  MoveL 5113 to (559.6, 473.58, 88) mm, rotated rx -180 ry 0 rz 160 deg; joints [2.536, 74.611, -25.018, -151.413, 53.222, 161.93]
  Set speed (17.9 mm/s)
  Call Extruder(373.72184)
  MoveL 5114 to (560.12, 474.8, 88) mm, rotated rx -180 ry 0 rz 160 deg; joints [2.67, 74.736, -25.273, -151.206, 53.149, 161.757]
  Set speed (17.9 mm/s)
  Call Extruder(378.01849)
  MoveL 5115 to (560.64, 476.06, 88) mm, rotated rx 180 ry 0 rz 160 deg; joints [2.809, 74.862, -25.532, -150.994, 53.077, 161.578]
  Set speed (17.9 mm/s)
  Call Extruder(382.11956)
  MoveL 5116 to (561.1, 477.28, 88) mm, rotated rx -180 ry 0 rz 160 deg; joints [2.943, 74.976, -25.765, -150.791, 53.016, 161.41]
  Set speed (17.9 mm/s)
  Call Extruder(386.18215)
  MoveL 5117 to (561.55, 478.49, 88) mm, rotated rx -180 ry 0 rz 160 deg; joints [3.076, 75.088, -25.993, -150.59, 52.957, 161.244]
  Call Extruder(390.52183)
  MoveL 5118 to (561.98, 479.8, 88) mm, rotated rx 180 ry 0 rz 160 deg; joints [3.219, 75.2, -26.222, -150.377, 52.902, 161.069]
  Set speed (17.9 mm/s)
  Call Extruder(394.64842)
  MoveL 5119 to (562.38, 481.05, 88) mm, rotated rx -180 ry 0 rz 160 deg; joints [3.356, 75.305, -26.435, -150.174, 52.852, 160.904]
  Set speed (17.9 mm/s)
  Call Extruder(398.90970)
  MoveL 5120 to (562.75, 482.35, 88) mm, rotated rx 180 ry 0 rz 160 deg; joints [3.499, 75.405, -26.64, -149.965, 52.808, 160.736]
  Set speed (17.9 mm/s)
  Call Extruder(402.92421)
  MoveL 5121 to (563.09, 483.58, 88) mm, rotated rx -180 ry 0 rz 160 deg; joints [3.633, 75.498, -26.83, -149.769, 52.769, 160.579]
  Call Extruder(407.31030)
  MoveL 5122 to (563.42, 484.93, 88) mm, rotated rx 180 ry 0 rz 160 deg; joints [3.781, 75.593, -27.022, -149.556, 52.735, 160.411]
  Set speed (17.9 mm/s)
  Call Extruder(411.41596)
  MoveL 5123 to (563.72, 486.2, 88) mm, rotated rx 180 ry 0 rz 160 deg; joints [3.92, 75.678, -27.196, -149.357, 52.705, 160.254]
  Set speed (17.9 mm/s)
  Call Extruder(419.87700)
  MoveL 5124 to (564.23, 488.84, 88) mm, rotated rx -180 ry 0 rz 160 deg; joints [4.21, 75.838, -27.52, -148.951, 52.662, 159.941]
  Set speed (17.9 mm/s)
  Call Extruder(428.25790)
  MoveL 5125 to (564.64, 491.48, 88) mm, rotated rx -180 ry 0 rz 160 deg; joints [4.499, 75.975, -27.801, -148.553, 52.64, 159.641]
  Call Extruder(436.73506)
  MoveL 5126 to (564.94, 494.16, 88) mm, rotated rx 180 ry 0 rz 160 deg; joints [4.793, 76.093, -28.041, -148.158, 52.639, 159.35]
  Call Extruder(445.02927)
  MoveL 5127 to (565.12, 496.79, 88) mm, rotated rx 180 ry 0 rz 160 deg; joints [5.082, 76.188, -28.232, -147.778, 52.659, 159.079]
  Call Extruder(453.41460)
  MoveL 5128 to (565.2, 499.45, 88) mm, rotated rx -180 ry 0 rz 160 deg; joints [5.376, 76.262, -28.384, -147.402, 52.7, 158.818]
  Set speed (18.0 mm/s)
  Call Extruder(461.67884)
  MoveL 5129 to (565.16, 502.08, 88) mm, rotated rx -180 ry 0 rz 160 deg; joints [5.666, 76.314, -28.488, -147.04, 52.761, 158.576]
  Set speed (17.9 mm/s)
  Call Extruder(470.17572)
  MoveL 5130 to (565.02, 504.78, 88) mm, rotated rx -180 ry 0 rz 160 deg; joints [5.965, 76.345, -28.551, -146.678, 52.844, 158.343]
  Call Extruder(478.48137)
  MoveL 5131 to (564.77, 507.41, 88) mm, rotated rx 180 ry 0 rz 160 deg; joints [6.258, 76.352, -28.566, -146.334, 52.946, 158.132]
  Set speed (18.0 mm/s)
  Call Extruder(487.03739)
  MoveL 5132 to (564.41, 510.11, 88) mm, rotated rx 180 ry 0 rz 160 deg; joints [6.559, 76.338, -28.536, -145.99, 53.071, 157.932]
  Call Extruder(495.31907)
  MoveL 5133 to (563.95, 512.71, 88) mm, rotated rx 180 ry 0 rz 160 deg; joints [6.851, 76.302, -28.464, -145.668, 53.212, 157.755]
  Set speed (17.9 mm/s)
  Call Extruder(503.76190)
  MoveL 5134 to (563.37, 515.33, 88) mm, rotated rx 180 ry 0 rz 160 deg; joints [7.147, 76.243, -28.344, -145.352, 53.374, 157.594]
  Set speed (17.9 mm/s)
  Call Extruder(507.92287)
  MoveL 5135 to (563.04, 516.61, 88) mm, rotated rx -180 ry 0 rz 160 deg; joints [7.293, 76.204, -28.266, -145.201, 53.463, 157.522]
  Set speed (17.9 mm/s)
  Call Extruder(512.03156)
  MoveL 5136 to (562.7, 517.87, 88) mm, rotated rx -180 ry 0 rz 160 deg; joints [7.436, 76.164, -28.183, -145.054, 53.552, 157.454]
  Set speed (17.9 mm/s)
  Call Extruder(516.36211)
  MoveL 5137 to (562.3, 519.18, 88) mm, rotated rx 180 ry 0 rz 160 deg; joints [7.587, 76.113, -28.08, -144.904, 53.653, 157.389]
  Set speed (17.9 mm/s)
  Call Extruder(520.51999)
  MoveL 5138 to (561.91, 520.44, 88) mm, rotated rx 180 ry 0 rz 160 deg; joints [7.731, 76.061, -27.975, -144.76, 53.752, 157.329]
  Set speed (17.9 mm/s)
  Call Extruder(528.91386)
  MoveL 5139 to (561.02, 522.96, 88) mm, rotated rx 180 ry 0 rz 160 deg; joints [8.022, 75.938, -27.725, -144.482, 53.968, 157.224]
  Set speed (17.9 mm/s)
  Call Extruder(533.10830)
  MoveL 5140 to (560.53, 524.2, 88) mm, rotated rx -180 ry 0 rz 160 deg; joints [8.166, 75.868, -27.582, -144.349, 54.083, 157.18]
  Set speed (17.9 mm/s)
  Call Extruder(537.31700)
  MoveL 5141 to (560.03, 525.44, 88) mm, rotated rx -180 ry 0 rz 160 deg; joints [8.311, 75.795, -27.433, -144.216, 54.2, 157.138]
  Set speed (17.9 mm/s)
  Call Extruder(541.50408)
  MoveL 5142 to (559.49, 526.66, 88) mm, rotated rx 180 ry 0 rz 160 deg; joints [8.453, 75.714, -27.269, -144.09, 54.323, 157.104]
  Set speed (17.9 mm/s)
  Call Extruder(545.52808)
  MoveL 5143 to (558.96, 527.82, 88) mm, rotated rx 180 ry 0 rz 160 deg; joints [8.59, 75.635, -27.107, -143.969, 54.443, 157.073]
  Set speed (17.9 mm/s)
  Call Extruder(548.70706)
  MoveL 5144 to (558.53, 528.73, 88) mm, rotated rx 180 ry 0 rz 160 deg; joints [8.698, 75.568, -26.972, -143.876, 54.541, 157.052]
  Set speed (17.9 mm/s)
  Call Extruder(554.38655)
  MoveL 5145 to (557.71, 530.34, 88) mm, rotated rx 180 ry 0 rz 160 deg; joints [8.889, 75.442, -26.714, -143.715, 54.721, 157.022]
  Set speed (18.0 mm/s)
  Call Extruder(558.28991)
  MoveL 5146 to (557.12, 531.43, 88) mm, rotated rx -180 ry 0 rz 160 deg; joints [9.02, 75.349, -26.526, -143.608, 54.85, 157.007]
  Set speed (17.9 mm/s)
  Call Extruder(562.42698)
  MoveL 5147 to (556.47, 532.58, 88) mm, rotated rx -180 ry 0 rz 160 deg; joints [9.158, 75.248, -26.319, -143.497, 54.989, 156.994]
  Set speed (18.0 mm/s)
  Call Extruder(566.58221)
  MoveL 5148 to (555.8, 533.72, 88) mm, rotated rx -180 ry 0 rz 160 deg; joints [9.296, 75.141, -26.102, -143.388, 55.131, 156.986]
  Call Extruder(570.79001)
  MoveL 5149 to (555.1, 534.86, 88) mm, rotated rx -180 ry 0 rz 160 deg; joints [9.435, 75.028, -25.872, -143.281, 55.28, 156.982]
  Set speed (17.9 mm/s)
  Call Extruder(574.99054)
  MoveL 5150 to (554.37, 535.98, 88) mm, rotated rx 180 ry 0 rz 160 deg; joints [9.572, 74.912, -25.633, -143.178, 55.431, 156.984]
  Set speed (17.9 mm/s)
  Call Extruder(579.19251)
  MoveL 5151 to (553.62, 537.08, 88) mm, rotated rx 180 ry 0 rz 160 deg; joints [9.709, 74.791, -25.387, -143.077, 55.585, 156.989]
  Set speed (17.9 mm/s)
  Call Extruder(583.43346)
  MoveL 5152 to (552.85, 538.19, 88) mm, rotated rx 180 ry 0 rz 160 deg; joints [9.846, 74.665, -25.129, -142.979, 55.744, 156.999]
  Call Extruder(587.57525)
  MoveL 5153 to (552.06, 539.24, 88) mm, rotated rx -180 ry 0 rz 160 deg; joints [9.978, 74.537, -24.867, -142.886, 55.902, 157.013]
  Set speed (17.9 mm/s)
  Call Extruder(591.76685)
  MoveL 5154 to (551.25, 540.3, 88) mm, rotated rx 180 ry 0 rz 160 deg; joints [10.111, 74.405, -24.597, -142.794, 56.064, 157.031]
  Call Extruder(595.94820)
  MoveL 5155 to (550.42, 541.34, 88) mm, rotated rx 180 ry 0 rz 160 deg; joints [10.243, 74.268, -24.317, -142.707, 56.229, 157.054]
  Set speed (17.9 mm/s)
  Call Extruder(600.26743)
  MoveL 5156 to (549.53, 542.39, 88) mm, rotated rx 180 ry 0 rz 160 deg; joints [10.377, 74.124, -24.021, -142.619, 56.403, 157.082]
  Set speed (17.9 mm/s)
  Call Extruder(604.33296)
  MoveL 5157 to (548.68, 543.36, 88) mm, rotated rx 180 ry 0 rz 160 deg; joints [10.503, 73.984, -23.734, -142.539, 56.568, 157.113]
  Set speed (17.9 mm/s)
  Call Extruder(608.56191)
  MoveL 5158 to (547.78, 544.36, 88) mm, rotated rx 180 ry 0 rz 160 deg; joints [10.633, 73.835, -23.429, -142.459, 56.742, 157.148]
  Set speed (17.9 mm/s)
  Call Extruder(612.71555)
  MoveL 5159 to (546.87, 545.32, 88) mm, rotated rx -180 ry 0 rz 160 deg; joints [10.759, 73.686, -23.123, -142.383, 56.916, 157.187]
  Set speed (17.9 mm/s)
  Call Extruder(616.93142)
  MoveL 5160 to (545.93, 546.27, 88) mm, rotated rx 180 ry 0 rz 160 deg; joints [10.885, 73.531, -22.805, -142.309, 57.094, 157.23]
  Set speed (18.0 mm/s)
  Call Extruder(621.11476)
  MoveL 5161 to (544.98, 547.2, 88) mm, rotated rx 180 ry 0 rz 160 deg; joints [11.009, 73.374, -22.482, -142.238, 57.273, 157.277]
  Set speed (17.9 mm/s)
  Call Extruder(625.39673)
  MoveL 5162 to (543.98, 548.13, 88) mm, rotated rx 180 ry 0 rz 160 deg; joints [11.135, 73.21, -22.144, -142.168, 57.459, 157.329]
  Set speed (17.9 mm/s)
  Call Extruder(629.55539)
  MoveL 5163 to (543, 549.01, 88) mm, rotated rx -180 ry 0 rz 160 deg; joints [11.255, 73.048, -21.81, -142.104, 57.641, 157.383]
  Set speed (17.9 mm/s)
  Call Extruder(633.66255)
  MoveL 5164 to (542, 549.86, 88) mm, rotated rx 180 ry 0 rz 160 deg; joints [11.373, 72.885, -21.474, -142.042, 57.823, 157.44]
  Call Extruder(637.94036)
  MoveL 5165 to (540.96, 550.73, 88) mm, rotated rx 180 ry 0 rz 160 deg; joints [11.494, 72.712, -21.118, -141.981, 58.013, 157.503]
  Set speed (17.9 mm/s)
  Call Extruder(642.04901)
  MoveL 5166 to (539.93, 551.54, 88) mm, rotated rx 180 ry 0 rz 160 deg; joints [11.608, 72.544, -20.771, -141.925, 58.198, 157.567]
  Call Extruder(646.27944)
  MoveL 5167 to (538.86, 552.35, 88) mm, rotated rx 180 ry 0 rz 160 deg; joints [11.725, 72.368, -20.407, -141.87, 58.39, 157.637]
  Set speed (17.9 mm/s)
  Call Extruder(650.48406)
  MoveL 5168 to (537.78, 553.14, 88) mm, rotated rx -180 ry 0 rz 160 deg; joints [11.839, 72.191, -20.041, -141.818, 58.582, 157.709]
  Call Extruder(654.65527)
  MoveL 5169 to (536.69, 553.89, 88) mm, rotated rx 180 ry 0 rz 160 deg; joints [11.95, 72.013, -19.672, -141.769, 58.774, 157.785]
  Set speed (17.9 mm/s)
  Call Extruder(658.83011)
  MoveL 5170 to (535.58, 554.63, 88) mm, rotated rx 180 ry 0 rz 160 deg; joints [12.06, 71.832, -19.299, -141.723, 58.967, 157.863]
  Set speed (17.9 mm/s)
  Call Extruder(663.02238)
  MoveL 5171 to (534.46, 555.35, 88) mm, rotated rx 180 ry 0 rz 160 deg; joints [12.168, 71.649, -18.919, -141.679, 59.162, 157.945]
  Set speed (17.9 mm/s)
  Call Extruder(667.21459)
  MoveL 5172 to (533.32, 556.04, 88) mm, rotated rx -180 ry 0 rz 160 deg; joints [12.274, 71.464, -18.535, -141.638, 59.358, 158.03]
  Set speed (18.0 mm/s)
  Call Extruder(671.40809)
  MoveL 5173 to (532.17, 556.71, 88) mm, rotated rx -180 ry 0 rz 160 deg; joints [12.379, 71.276, -18.145, -141.599, 59.556, 158.118]
  Set speed (17.9 mm/s)
  Call Extruder(675.05317)
  MoveL 5174 to (531.15, 557.28, 88) mm, rotated rx 180 ry 0 rz 160 deg; joints [12.468, 71.112, -17.804, -141.567, 59.728, 158.197]
  Set speed (17.9 mm/s)
  Call Extruder(679.85489)
  MoveL 5175 to (529.8, 557.99, 88) mm, rotated rx -180 ry 0 rz 160 deg; joints [12.584, 70.894, -17.349, -141.529, 59.955, 158.305]
  Set speed (17.9 mm/s)
  Call Extruder(684.04696)
  MoveL 5176 to (528.61, 558.59, 88) mm, rotated rx -180 ry 0 rz 160 deg; joints [12.682, 70.701, -16.948, -141.498, 60.155, 158.402]
  Set speed (17.9 mm/s)
  Call Extruder(688.17169)
  MoveL 5177 to (527.43, 559.15, 88) mm, rotated rx -180 ry 0 rz 160 deg; joints [12.777, 70.51, -16.55, -141.47, 60.352, 158.5]
  Set speed (17.9 mm/s)
  Call Extruder(692.46193)
  MoveL 5178 to (526.18, 559.7, 88) mm, rotated rx -180 ry 0 rz 160 deg; joints [12.873, 70.31, -16.132, -141.444, 60.557, 158.606]
  Set speed (17.9 mm/s)
  Call Extruder(696.56563)
  MoveL 5179 to (524.99, 560.22, 88) mm, rotated rx -180 ry 0 rz 160 deg; joints [12.964, 70.118, -15.731, -141.421, 60.754, 158.708]
  Set speed (17.9 mm/s)
  Call Extruder(700.85853)
  MoveL 5180 to (523.72, 560.72, 88) mm, rotated rx -180 ry 0 rz 160 deg; joints [13.055, 69.915, -15.306, -141.4, 60.96, 158.819]
  Set speed (17.9 mm/s)
  Call Extruder(704.88381)
  MoveL 5181 to (522.52, 561.18, 88) mm, rotated rx -180 ry 0 rz 160 deg; joints [13.14, 69.725, -14.907, -141.382, 61.154, 158.924]
  Set speed (17.9 mm/s)
  Call Extruder(709.30941)
  MoveL 5182 to (521.2, 561.65, 88) mm, rotated rx -180 ry 0 rz 160 deg; joints [13.229, 69.513, -14.464, -141.366, 61.367, 159.043]
  Set speed (17.9 mm/s)
  Call Extruder(713.41630)
  MoveL 5183 to (519.97, 562.07, 88) mm, rotated rx 180 ry 0 rz 160 deg; joints [13.311, 69.317, -14.053, -141.352, 61.564, 159.154]
  Call Extruder(717.65007)
  MoveL 5184 to (518.68, 562.46, 88) mm, rotated rx -180 ry 0 rz 160 deg; joints [13.392, 69.113, -13.624, -141.342, 61.768, 159.273]
  Set speed (17.9 mm/s)
  Call Extruder(721.92491)
  MoveL 5185 to (517.38, 562.84, 88) mm, rotated rx -180 ry 0 rz 160 deg; joints [13.472, 68.907, -13.191, -141.332, 61.974, 159.394]
  Set speed (17.9 mm/s)
  Call Extruder(725.52012)
  MoveL 5186 to (516.27, 563.13, 88) mm, rotated rx -180 ry 0 rz 160 deg; joints [13.537, 68.733, -12.823, -141.328, 62.148, 159.498]
  Set speed (17.9 mm/s)
  Call Extruder(730.10548)
  MoveL 5187 to (514.86, 563.48, 88) mm, rotated rx 180 ry 0 rz 160 deg; joints [13.618, 68.511, -12.355, -141.323, 62.368, 159.632]
  Set speed (17.9 mm/s)
  Call Extruder(738.64656)
  MoveL 5188 to (512.2, 564.04, 88) mm, rotated rx -180 ry 0 rz 160 deg; joints [13.759, 68.094, -11.474, -141.324, 62.779, 159.89]
  Set speed (17.9 mm/s)
  Call Extruder(747.08753)
  MoveL 5189 to (509.56, 564.49, 88) mm, rotated rx 180 ry 0 rz 160 deg; joints [13.888, 67.681, -10.599, -141.335, 63.184, 160.152]
  Call Extruder(755.39717)
  MoveL 5190 to (506.93, 564.83, 88) mm, rotated rx 180 ry 0 rz 160 deg; joints [14.004, 67.273, -9.734, -141.356, 63.58, 160.417]
  Set speed (17.9 mm/s)
  Call Extruder(763.82579)
  MoveL 5191 to (504.26, 565.06, 88) mm, rotated rx 180 ry 0 rz 160 deg; joints [14.111, 66.86, -8.855, -141.388, 63.98, 160.692]
  Set speed (18.0 mm/s)
  Call Extruder(772.24871)
  MoveL 5192 to (501.59, 565.18, 88) mm, rotated rx -180 ry 0 rz 160 deg; joints [14.206, 66.448, -7.974, -141.429, 64.377, 160.973]
  Set speed (17.9 mm/s)
  Call Extruder(780.47163)
  MoveL 5193 to (498.97, 565.19, 88) mm, rotated rx 180 ry 0 rz 160 deg; joints [14.286, 66.046, -7.115, -141.48, 64.761, 161.252]
  Set speed (10.0 mm/s)
  MoveL 5194 to (498.97, 565.19, 92) mm, rotated rx 180 ry 0 rz 160 deg; joints [14.286, 65.4, -6.792, -141.385, 64.508, 161.029]
  Set speed (120.0 mm/s)
  MoveL 5195 to (498.97, 565.42, 92) mm, rotated rx 180 ry 0 rz 160 deg; joints [14.315, 65.408, -6.81, -141.352, 64.51, 161.01]
  Set speed (18.0 mm/s)
  Call Extruder(789.01663)
  MoveL 5196 to (496.25, 565.32, 92) mm, rotated rx 180 ry 0 rz 160 deg; joints [14.386, 64.991, -5.919, -141.417, 64.903, 161.305]
  Call Extruder(797.44924)
  MoveL 5197 to (493.57, 565.11, 92) mm, rotated rx 180 ry 0 rz 160 deg; joints [14.444, 64.581, -5.043, -141.491, 65.286, 161.6]
  Set speed (18.0 mm/s)
  Call Extruder(805.77515)
  MoveL 5198 to (490.93, 564.8, 92) mm, rotated rx -180 ry 0 rz 160 deg; joints [14.489, 64.18, -4.182, -141.575, 65.66, 161.895]
  Set speed (18.0 mm/s)
  Call Extruder(814.13501)
  MoveL 5199 to (488.31, 564.38, 92) mm, rotated rx -180 ry 0 rz 160 deg; joints [14.52, 63.78, -3.323, -141.67, 66.031, 162.194]
  Set speed (18.0 mm/s)
  Call Extruder(822.67375)
  MoveL 5200 to (485.64, 563.84, 92) mm, rotated rx 180 ry 0 rz 160 deg; joints [14.539, 63.376, -2.451, -141.779, 66.403, 162.503]
  Set speed (18.0 mm/s)
  Call Extruder(826.82258)
  MoveL 5201 to (484.36, 563.53, 92) mm, rotated rx 180 ry 0 rz 160 deg; joints [14.542, 63.182, -2.031, -141.837, 66.582, 162.654]
  Set speed (17.9 mm/s)
  Call Extruder(831.03549)
  MoveL 5202 to (483.06, 563.2, 92) mm, rotated rx 180 ry 0 rz 160 deg; joints [14.543, 62.986, -1.607, -141.896, 66.762, 162.807]
  Set speed (18.0 mm/s)
  Call Extruder(835.18857)
  MoveL 5203 to (481.79, 562.84, 92) mm, rotated rx 180 ry 0 rz 160 deg; joints [14.539, 62.794, -1.19, -141.96, 66.937, 162.959]
  Call Extruder(839.32320)
  MoveL 5204 to (480.52, 562.47, 92) mm, rotated rx 180 ry 0 rz 160 deg; joints [14.533, 62.604, -0.778, -142.023, 67.111, 163.11]
  Call Extruder(843.60530)
  MoveL 5205 to (479.23, 562.04, 92) mm, rotated rx 180 ry 0 rz 160 deg; joints [14.522, 62.409, -0.353, -142.094, 67.289, 163.268]
  Set speed (18.0 mm/s)
  Call Extruder(847.72562)
  MoveL 5206 to (477.99, 561.62, 92) mm, rotated rx -180 ry 0 rz 160 deg; joints [14.509, 62.222, 0.053, -142.164, 67.458, 163.419]
  Call Extruder(852.06033)
  MoveL 5207 to (476.7, 561.13, 92) mm, rotated rx -180 ry 0 rz 160 deg; joints [14.491, 62.028, 0.478, -142.242, 67.635, 163.579]
  Set speed (18.0 mm/s)
  Call Extruder(856.17794)
  MoveL 5208 to (475.48, 560.66, 92) mm, rotated rx -180 ry 0 rz 160 deg; joints [14.471, 61.845, 0.878, -142.317, 67.801, 163.73]
  Set speed (17.9 mm/s)
  Call Extruder(858.47099)
  MoveL 5209 to (474.8, 560.38, 92) mm, rotated rx 180 ry 0 rz 160 deg; joints [14.458, 61.743, 1.1, -142.36, 67.892, 163.815]
  Set speed (17.9 mm/s)
  Call Extruder(864.46055)
  MoveL 5210 to (473.05, 559.62, 92) mm, rotated rx -180 ry 0 rz 160 deg; joints [14.418, 61.481, 1.674, -142.478, 68.129, 164.036]
  Set speed (18.0 mm/s)
  Call Extruder(868.83195)
  MoveL 5211 to (471.79, 559.04, 92) mm, rotated rx 180 ry 0 rz 160 deg; joints [14.385, 61.291, 2.091, -142.567, 68.3, 164.197]
  Set speed (18.0 mm/s)
  Call Extruder(873.01855)
  MoveL 5212 to (470.59, 558.45, 92) mm, rotated rx 180 ry 0 rz 160 deg; joints [14.349, 61.112, 2.485, -142.657, 68.461, 164.351]
  Set speed (18.0 mm/s)
  Call Extruder(875.99211)
  MoveL 5213 to (469.75, 558.02, 92) mm, rotated rx -180 ry 0 rz 160 deg; joints [14.322, 60.985, 2.764, -142.721, 68.574, 164.461]
  Set speed (18.0 mm/s)
  Call Extruder(881.36896)
  MoveL 5214 to (468.24, 557.21, 92) mm, rotated rx -180 ry 0 rz 160 deg; joints [14.266, 60.759, 3.262, -142.843, 68.777, 164.658]
  Set speed (18.0 mm/s)
  Call Extruder(885.56073)
  MoveL 5215 to (467.08, 556.55, 92) mm, rotated rx -180 ry 0 rz 160 deg; joints [14.219, 60.585, 3.647, -142.941, 68.932, 164.812]
  Set speed (18.0 mm/s)
  Call Extruder(889.80771)
  MoveL 5216 to (465.92, 555.85, 92) mm, rotated rx 180 ry 0 rz 160 deg; joints [14.168, 60.411, 4.033, -143.043, 69.087, 164.967]
  Call Extruder(894.07530)
  MoveL 5217 to (464.76, 555.13, 92) mm, rotated rx 180 ry 0 rz 160 deg; joints [14.112, 60.238, 4.416, -143.149, 69.241, 165.123]
  Set speed (18.0 mm/s)
  Call Extruder(897.51102)
  MoveL 5218 to (463.85, 554.53, 92) mm, rotated rx -180 ry 0 rz 160 deg; joints [14.063, 60.1, 4.721, -143.236, 69.363, 165.248]
  Call Extruder(902.37563)
  MoveL 5219 to (462.57, 553.66, 92) mm, rotated rx -180 ry 0 rz 160 deg; joints [13.992, 59.907, 5.149, -143.363, 69.534, 165.424]
  Set speed (18.0 mm/s)
  Call Extruder(906.61401)
  MoveL 5220 to (461.47, 552.88, 92) mm, rotated rx -180 ry 0 rz 160 deg; joints [13.925, 59.742, 5.517, -143.477, 69.68, 165.577]
  Set speed (18.0 mm/s)
  Call Extruder(910.79311)
  MoveL 5221 to (460.4, 552.08, 92) mm, rotated rx -180 ry 0 rz 160 deg; joints [13.855, 59.582, 5.875, -143.593, 69.821, 165.727]
  Set speed (18.0 mm/s)
  Call Extruder(914.94843)
  MoveL 5222 to (459.35, 551.27, 92) mm, rotated rx 180 ry 0 rz 160 deg; joints [13.782, 59.424, 6.227, -143.711, 69.959, 165.876]
  Set speed (18.0 mm/s)
  Call Extruder(919.19020)
  MoveL 5223 to (458.3, 550.42, 92) mm, rotated rx 180 ry 0 rz 160 deg; joints [13.703, 59.266, 6.581, -143.834, 70.098, 166.027]
  Set speed (18.0 mm/s)
  Call Extruder(923.41678)
  MoveL 5224 to (457.27, 549.55, 92) mm, rotated rx 180 ry 0 rz 160 deg; joints [13.62, 59.111, 6.928, -143.96, 70.234, 166.176]
  Set speed (18.0 mm/s)
  Call Extruder(927.58466)
  MoveL 5225 to (456.27, 548.67, 92) mm, rotated rx 180 ry 0 rz 160 deg; joints [13.536, 58.96, 7.266, -144.087, 70.365, 166.322]
  Set speed (18.0 mm/s)
  Call Extruder(932.62885)
  MoveL 5226 to (455.09, 547.59, 92) mm, rotated rx 180 ry 0 rz 160 deg; joints [13.428, 58.781, 7.669, -144.244, 70.521, 166.498]
  Call Extruder(935.97678)
  MoveL 5227 to (454.32, 546.85, 92) mm, rotated rx 180 ry 0 rz 160 deg; joints [13.353, 58.664, 7.931, -144.351, 70.622, 166.614]
  Set speed (18.0 mm/s)
  Call Extruder(940.18635)
  MoveL 5228 to (453.37, 545.9, 92) mm, rotated rx -180 ry 0 rz 160 deg; joints [13.256, 58.52, 8.257, -144.488, 70.747, 166.759]
  Call Extruder(944.36556)
  MoveL 5229 to (452.45, 544.94, 92) mm, rotated rx -180 ry 0 rz 160 deg; joints [13.156, 58.379, 8.574, -144.627, 70.868, 166.901]
  Set speed (18.0 mm/s)
  Call Extruder(949.38745)
  MoveL 5230 to (451.36, 543.77, 92) mm, rotated rx 180 ry 0 rz 160 deg; joints [13.031, 58.214, 8.948, -144.798, 71.01, 167.071]
  Set speed (18.0 mm/s)
  Call Extruder(956.56674)
  MoveL 5231 to (449.86, 542.04, 92) mm, rotated rx 180 ry 0 rz 160 deg; joints [12.843, 57.984, 9.468, -145.048, 71.206, 167.31]
  Set speed (18.0 mm/s)
  Call Extruder(961.19648)
  MoveL 5232 to (448.93, 540.9, 92) mm, rotated rx 180 ry 0 rz 160 deg; joints [12.716, 57.841, 9.794, -145.215, 71.329, 167.462]
  Set speed (18.0 mm/s)
  Call Extruder(965.38017)
  MoveL 5233 to (448.11, 539.85, 92) mm, rotated rx 180 ry 0 rz 160 deg; joints [12.598, 57.714, 10.082, -145.368, 71.436, 167.598]
  Set speed (18.0 mm/s)
  Call Extruder(969.61345)
  MoveL 5234 to (447.3, 538.77, 92) mm, rotated rx -180 ry 0 rz 160 deg; joints [12.474, 57.589, 10.368, -145.525, 71.541, 167.735]
  Call Extruder(973.80355)
  MoveL 5235 to (446.52, 537.69, 92) mm, rotated rx -180 ry 0 rz 160 deg; joints [12.348, 57.467, 10.645, -145.684, 71.643, 167.868]
  Set speed (18.0 mm/s)
  Call Extruder(978.00195)
  MoveL 5236 to (445.76, 536.59, 92) mm, rotated rx 180 ry 0 rz 160 deg; joints [12.219, 57.349, 10.915, -145.846, 71.741, 168]
  Set speed (18.0 mm/s)
  Call Extruder(982.22074)
  MoveL 5237 to (445.02, 535.47, 92) mm, rotated rx 180 ry 0 rz 160 deg; joints [12.085, 57.233, 11.181, -146.011, 71.838, 168.131]
  Set speed (18.0 mm/s)
  Call Extruder(986.41735)
  MoveL 5238 to (444.3, 534.34, 92) mm, rotated rx -180 ry 0 rz 160 deg; joints [11.949, 57.12, 11.438, -146.178, 71.93, 168.26]
  Call Extruder(990.55322)
  MoveL 5239 to (443.62, 533.21, 92) mm, rotated rx -180 ry 0 rz 160 deg; joints [11.812, 57.013, 11.685, -146.344, 72.018, 168.385]
  Set speed (18.0 mm/s)
  Call Extruder(994.88630)
  MoveL 5240 to (442.94, 532.01, 92) mm, rotated rx 180 ry 0 rz 160 deg; joints [11.664, 56.903, 11.936, -146.522, 72.107, 168.514]
  Call Extruder(998.92743)
  MoveL 5241 to (442.32, 530.88, 92) mm, rotated rx 180 ry 0 rz 160 deg; joints [11.524, 56.804, 12.164, -146.689, 72.186, 168.633]
  Set speed (18.0 mm/s)
  Call Extruder(1003.20251)
  MoveL 5242 to (441.69, 529.68, 92) mm, rotated rx 180 ry 0 rz 160 deg; joints [11.372, 56.702, 12.399, -146.869, 72.268, 168.757]
  Set speed (18.0 mm/s)
  Call Extruder(1007.35394)
  MoveL 5243 to (441.1, 528.49, 92) mm, rotated rx 180 ry 0 rz 160 deg; joints [11.222, 56.606, 12.62, -147.045, 72.343, 168.876]
  Set speed (18.0 mm/s)
  Call Extruder(1015.72244)
  MoveL 5244 to (439.99, 526.07, 92) mm, rotated rx 180 ry 0 rz 160 deg; joints [10.909, 56.423, 13.043, -147.408, 72.485, 169.109]
  Set speed (17.9 mm/s)
  Call Extruder(1020.10838)
  MoveL 5245 to (439.45, 524.78, 92) mm, rotated rx 180 ry 0 rz 160 deg; joints [10.741, 56.333, 13.251, -147.601, 72.553, 169.228]
  Call Extruder(1024.19326)
  MoveL 5246 to (438.96, 523.58, 92) mm, rotated rx 180 ry 0 rz 160 deg; joints [10.582, 56.251, 13.441, -147.783, 72.615, 169.337]
  Call Extruder(1028.49518)
  MoveL 5247 to (438.49, 522.29, 92) mm, rotated rx -180 ry 0 rz 160 deg; joints [10.412, 56.17, 13.63, -147.977, 72.674, 169.449]
  Call Extruder(1032.65584)
  MoveL 5248 to (438.05, 521.05, 92) mm, rotated rx -180 ry 0 rz 160 deg; joints [10.245, 56.093, 13.808, -148.165, 72.73, 169.557]
  Call Extruder(1036.92105)
  MoveL 5249 to (437.63, 519.76, 92) mm, rotated rx 180 ry 0 rz 160 deg; joints [10.07, 56.019, 13.98, -148.361, 72.782, 169.664]
  Set speed (18.0 mm/s)
  Call Extruder(1041.13480)
  MoveL 5250 to (437.23, 518.48, 92) mm, rotated rx 180 ry 0 rz 160 deg; joints [9.896, 55.948, 14.145, -148.555, 72.831, 169.768]
  Set speed (18.0 mm/s)
  Call Extruder(1045.34721)
  MoveL 5251 to (436.87, 517.18, 92) mm, rotated rx 180 ry 0 rz 160 deg; joints [9.719, 55.882, 14.299, -148.752, 72.875, 169.87]
  Set speed (18.0 mm/s)
  Call Extruder(1049.40418)
  MoveL 5252 to (436.54, 515.94, 92) mm, rotated rx -180 ry 0 rz 160 deg; joints [9.547, 55.82, 14.443, -148.942, 72.915, 169.966]
  Set speed (17.9 mm/s)
  Call Extruder(1053.14225)
  MoveL 5253 to (436.27, 514.78, 92) mm, rotated rx 180 ry 0 rz 160 deg; joints [9.387, 55.767, 14.566, -149.118, 72.948, 170.053]
  Call Extruder(1058.14576)
  MoveL 5254 to (435.92, 513.23, 92) mm, rotated rx 180 ry 0 rz 160 deg; joints [9.17, 55.699, 14.725, -149.356, 72.988, 170.167]
  Set speed (18.0 mm/s)
  Call Extruder(1066.38434)
  MoveL 5255 to (435.44, 510.65, 92) mm, rotated rx -180 ry 0 rz 160 deg; joints [8.806, 55.599, 14.958, -149.751, 73.042, 170.347]
  Set speed (18.0 mm/s)
  Call Extruder(1074.77639)
  MoveL 5256 to (435.06, 508, 92) mm, rotated rx 180 ry 0 rz 160 deg; joints [8.429, 55.511, 15.164, -150.158, 73.081, 170.522]
  Set speed (18.0 mm/s)
  Call Extruder(1083.18865)
  MoveL 5257 to (434.79, 505.33, 92) mm, rotated rx -180 ry 0 rz 160 deg; joints [8.046, 55.437, 15.338, -150.568, 73.105, 170.688]
  Set speed (18.0 mm/s)
  Call Extruder(1091.42334)
  MoveL 5258 to (434.63, 502.71, 92) mm, rotated rx -180 ry 0 rz 160 deg; joints [7.666, 55.378, 15.475, -150.972, 73.113, 170.842]
  Set speed (18.0 mm/s)
  Call Extruder(1099.90321)
  MoveL 5259 to (434.57, 500.01, 92) mm, rotated rx 180 ry 0 rz 160 deg; joints [7.27, 55.332, 15.583, -151.389, 73.105, 170.992]
  Call Extruder(1107.54449)
  MoveL 5260 to (434.62, 497.58, 92) mm, rotated rx -180 ry 0 rz 160 deg; joints [6.912, 55.303, 15.651, -151.765, 73.083, 171.119]
  Set speed (18.0 mm/s)
  Call Extruder(1114.96621)
  MoveL 5261 to (434.74, 495.22, 92) mm, rotated rx 180 ry 0 rz 160 deg; joints [6.562, 55.287, 15.69, -152.129, 73.049, 171.235]
  Set speed (18.0 mm/s)
  Call Extruder(1122.51883)
  MoveL 5262 to (434.97, 492.82, 92) mm, rotated rx -180 ry 0 rz 160 deg; joints [6.206, 55.281, 15.703, -152.499, 73.002, 171.347]
  Call Extruder(1130.15594)
  MoveL 5263 to (435.28, 490.41, 92) mm, rotated rx 180 ry 0 rz 160 deg; joints [5.845, 55.288, 15.687, -152.871, 72.94, 171.452]
  Set speed (18.0 mm/s)
  Call Extruder(1137.79824)
  MoveL 5264 to (435.68, 488.01, 92) mm, rotated rx 180 ry 0 rz 160 deg; joints [5.485, 55.306, 15.645, -153.24, 72.865, 171.549]
  Call Extruder(1145.20707)
  MoveL 5265 to (436.15, 485.7, 92) mm, rotated rx -180 ry 0 rz 160 deg; joints [5.138, 55.335, 15.576, -153.594, 72.779, 171.637]
  Call Extruder(1152.69209)
  MoveL 5266 to (436.72, 483.38, 92) mm, rotated rx -180 ry 0 rz 160 deg; joints [4.789, 55.376, 15.48, -153.948, 72.679, 171.719]
  Call Extruder(1160.29922)
  MoveL 5267 to (437.38, 481.05, 92) mm, rotated rx 180 ry 0 rz 160 deg; joints [4.437, 55.429, 15.356, -154.302, 72.565, 171.795]
  Set speed (18.0 mm/s)
  Call Extruder(1167.89288)
  MoveL 5268 to (438.12, 478.75, 92) mm, rotated rx -180 ry 0 rz 160 deg; joints [4.09, 55.494, 15.204, -154.651, 72.437, 171.864]
  Set speed (18.0 mm/s)
  Call Extruder(1175.51580)
  MoveL 5269 to (438.95, 476.46, 92) mm, rotated rx -180 ry 0 rz 160 deg; joints [3.746, 55.571, 15.025, -154.994, 72.295, 171.927]
  Set speed (18.0 mm/s)
  Call Extruder(1182.28934)
  MoveL 5270 to (439.76, 474.46, 92) mm, rotated rx 180 ry 0 rz 160 deg; joints [3.445, 55.648, 14.843, -155.293, 72.159, 171.976]
  Set speed (18.0 mm/s)
  Call Extruder(1190.64289)
  MoveL 5271 to (440.85, 472.04, 92) mm, rotated rx 180 ry 0 rz 160 deg; joints [3.08, 55.757, 14.59, -155.654, 71.976, 172.03]
  Set speed (18.0 mm/s)
  Call Extruder(1198.29599)
  MoveL 5272 to (441.93, 469.85, 92) mm, rotated rx 180 ry 0 rz 160 deg; joints [2.753, 55.868, 14.33, -155.975, 71.796, 172.072]
  Set speed (18.0 mm/s)
  Call Extruder(1205.76517)
  MoveL 5273 to (443.06, 467.76, 92) mm, rotated rx -180 ry 0 rz 160 deg; joints [2.44, 55.988, 14.05, -156.28, 71.607, 172.107]
  Call Extruder(1213.40735)
  MoveL 5274 to (444.3, 465.66, 92) mm, rotated rx 180 ry 0 rz 160 deg; joints [2.127, 56.122, 13.74, -156.583, 71.402, 172.136]
  Set speed (18.0 mm/s)
  Call Extruder(1220.88255)
  MoveL 5275 to (445.59, 463.66, 92) mm, rotated rx 180 ry 0 rz 160 deg; joints [1.83, 56.264, 13.411, -156.869, 71.19, 172.158]
  Call Extruder(1228.43806)
  MoveL 5276 to (446.96, 461.68, 92) mm, rotated rx 180 ry 0 rz 160 deg; joints [1.538, 56.418, 13.055, -157.148, 70.964, 172.173]
  Set speed (18.0 mm/s)
  Call Extruder(1236.07803)
  MoveL 5277 to (448.43, 459.74, 92) mm, rotated rx 180 ry 0 rz 160 deg; joints [1.252, 56.584, 12.671, -157.418, 70.724, 172.183]
  Call Extruder(1243.56314)
  MoveL 5278 to (449.93, 457.88, 92) mm, rotated rx -180 ry 0 rz 160 deg; joints [0.982, 56.758, 12.271, -157.672, 70.478, 172.185]
  Set speed (18.0 mm/s)
  Call Extruder(1251.11719)
  MoveL 5279 to (451.51, 456.07, 92) mm, rotated rx -180 ry 0 rz 160 deg; joints [0.718, 56.943, 11.845, -157.916, 70.219, 172.182]
  Call Extruder(1258.75501)
  MoveL 5280 to (453.18, 454.3, 92) mm, rotated rx -180 ry 0 rz 160 deg; joints [0.463, 57.141, 11.391, -158.151, 69.947, 172.172]
  Call Extruder(1266.22751)
  MoveL 5281 to (454.87, 452.62, 92) mm, rotated rx -180 ry 0 rz 160 deg; joints [0.224, 57.344, 10.925, -158.367, 69.671, 172.155]
  Call Extruder(1273.78413)
  MoveL 5282 to (456.65, 450.99, 92) mm, rotated rx 180 ry 0 rz 160 deg; joints [-0.007, 57.559, 10.434, -158.574, 69.383, 172.133]
  Set speed (18.0 mm/s)
  Call Extruder(1281.16786)
  MoveL 5283 to (458.44, 449.47, 92) mm, rotated rx 180 ry 0 rz 160 deg; joints [-0.221, 57.779, 9.934, -158.762, 69.092, 172.104]
  Set speed (18.0 mm/s)
  Call Extruder(1289.14229)
  MoveL 5284 to (460.43, 447.89, 92) mm, rotated rx -180 ry 0 rz 160 deg; joints [-0.441, 58.026, 9.374, -158.952, 68.769, 172.066]
  Set speed (18.0 mm/s)
  Call Extruder(1296.00615)
  MoveL 5285 to (462.19, 446.6, 92) mm, rotated rx -180 ry 0 rz 160 deg; joints [-0.619, 58.247, 8.874, -159.102, 68.484, 172.028]
  Call Extruder(1304.05043)
  MoveL 5286 to (464.31, 445.16, 92) mm, rotated rx -180 ry 0 rz 160 deg; joints [-0.815, 58.515, 8.269, -159.263, 68.142, 171.976]
  Set speed (18.0 mm/s)
  Call Extruder(1311.69781)
  MoveL 5287 to (466.37, 443.87, 92) mm, rotated rx -180 ry 0 rz 160 deg; joints [-0.989, 58.778, 7.675, -159.401, 67.808, 171.92]
  Set speed (18.0 mm/s)
  Call Extruder(1319.25394)
  MoveL 5288 to (468.46, 442.67, 92) mm, rotated rx 180 ry 0 rz 160 deg; joints [-1.148, 59.048, 7.07, -159.524, 67.471, 171.858]
  Set speed (18.0 mm/s)
  Call Extruder(1326.63480)
  MoveL 5289 to (470.54, 441.58, 92) mm, rotated rx 180 ry 0 rz 160 deg; joints [-1.292, 59.319, 6.462, -159.629, 67.136, 171.79]
  Call Extruder(1334.37561)
  MoveL 5290 to (472.77, 440.51, 92) mm, rotated rx 180 ry 0 rz 160 deg; joints [-1.43, 59.611, 5.81, -159.724, 66.778, 171.712]
  Set speed (18.0 mm/s)
  Call Extruder(1341.93230)
  MoveL 5291 to (474.97, 439.54, 92) mm, rotated rx 180 ry 0 rz 160 deg; joints [-1.553, 59.904, 5.158, -159.803, 66.423, 171.629]
  Set speed (18.0 mm/s)
  Call Extruder(1349.31857)
  MoveL 5292 to (477.16, 438.68, 92) mm, rotated rx -180 ry 0 rz 160 deg; joints [-1.66, 60.197, 4.506, -159.865, 66.071, 171.541]
  Set speed (18.0 mm/s)
  Call Extruder(1357.02805)
  MoveL 5293 to (479.48, 437.87, 92) mm, rotated rx -180 ry 0 rz 160 deg; joints [-1.76, 60.51, 3.813, -159.914, 65.699, 171.442]
  Set speed (18.0 mm/s)
  Call Extruder(1364.47266)
  MoveL 5294 to (481.75, 437.17, 92) mm, rotated rx -180 ry 0 rz 160 deg; joints [-1.844, 60.819, 3.13, -159.947, 65.336, 171.339]
  Set speed (18.0 mm/s)
  Call Extruder(1371.96815)
  MoveL 5295 to (484.05, 436.55, 92) mm, rotated rx -180 ry 0 rz 160 deg; joints [-1.916, 61.136, 2.431, -159.965, 64.966, 171.228]
  Set speed (18.0 mm/s)
  Call Extruder(1379.73436)
  MoveL 5296 to (486.46, 435.99, 92) mm, rotated rx 180 ry 0 rz 160 deg; joints [-1.979, 61.472, 1.695, -159.969, 64.58, 171.105]
  Set speed (18.0 mm/s)
  Call Extruder(1387.14760)
  MoveL 5297 to (488.78, 435.54, 92) mm, rotated rx 180 ry 0 rz 160 deg; joints [-2.027, 61.798, 0.981, -159.958, 64.208, 170.981]
  Set speed (18.0 mm/s)
  Call Extruder(1394.54313)
  MoveL 5298 to (491.11, 435.17, 92) mm, rotated rx -180 ry 0 rz 160 deg; joints [-2.064, 62.128, 0.26, -159.933, 63.835, 170.849]
  Set speed (18.0 mm/s)
  Call Extruder(1402.32020)
  MoveL 5299 to (493.57, 434.89, 92) mm, rotated rx 180 ry 0 rz 160 deg; joints [-2.089, 62.48, -0.507, -159.89, 63.441, 170.703]
  Set speed (18.0 mm/s)
  Call Extruder(1409.82233)
  MoveL 5300 to (495.95, 434.7, 92) mm, rotated rx 180 ry 0 rz 160 deg; joints [-2.103, 62.824, -1.256, -159.835, 63.059, 170.554]
  Call Extruder(1417.53399)
  MoveL 5301 to (498.41, 434.59, 92) mm, rotated rx 180 ry 0 rz 160 deg; joints [-2.105, 63.183, -2.033, -159.763, 62.666, 170.392]
  Set speed (18.0 mm/s)
  Call Extruder(1425.01271)
  MoveL 5302 to (500.79, 434.57, 92) mm, rotated rx -180 ry 0 rz 160 deg; joints [-2.096, 63.535, -2.793, -159.679, 62.285, 170.228]
  Call Extruder(1432.64222)
  MoveL 5303 to (503.23, 434.65, 92) mm, rotated rx 180 ry 0 rz 160 deg; joints [-2.075, 63.897, -3.574, -159.579, 61.896, 170.052]
  Set speed (18.0 mm/s)
  Call Extruder(1440.11283)
  MoveL 5304 to (505.6, 434.81, 92) mm, rotated rx 180 ry 0 rz 160 deg; joints [-2.044, 64.255, -4.343, -159.467, 61.516, 169.872]
  Set speed (18.0 mm/s)
  Call Extruder(1447.55032)
  MoveL 5305 to (507.96, 435.06, 92) mm, rotated rx 180 ry 0 rz 160 deg; joints [-2.002, 64.614, -5.113, -159.341, 61.139, 169.685]
  Set speed (18.0 mm/s)
  Call Extruder(1455.18005)
  MoveL 5306 to (510.36, 435.4, 92) mm, rotated rx -180 ry 0 rz 160 deg; joints [-1.95, 64.984, -5.906, -159.199, 60.753, 169.485]
  Set speed (18.0 mm/s)
  Call Extruder(1462.80028)
  MoveL 5307 to (512.75, 435.83, 92) mm, rotated rx -180 ry 0 rz 160 deg; joints [-1.886, 65.356, -6.7, -159.043, 60.371, 169.278]
  Set speed (18.0 mm/s)
  Call Extruder(1469.79314)
  MoveL 5308 to (514.93, 436.3, 92) mm, rotated rx 180 ry 0 rz 160 deg; joints [-1.82, 65.699, -7.43, -158.888, 60.022, 169.08]
  Set speed (18.0 mm/s)
  Call Extruder(1477.93243)
  MoveL 5309 to (517.44, 436.94, 92) mm, rotated rx 180 ry 0 rz 160 deg; joints [-1.731, 66.099, -8.279, -158.693, 59.619, 168.841]
  Set speed (18.0 mm/s)
  Call Extruder(1485.49614)
  MoveL 5310 to (519.75, 437.62, 92) mm, rotated rx -180 ry 0 rz 160 deg; joints [-1.639, 66.472, -9.069, -158.498, 59.249, 168.611]
  Call Extruder(1493.12816)
  MoveL 5311 to (522.06, 438.4, 92) mm, rotated rx 180 ry 0 rz 160 deg; joints [-1.537, 66.848, -9.865, -158.288, 58.88, 168.371]
  Call Extruder(1500.60168)
  MoveL 5312 to (524.28, 439.24, 92) mm, rotated rx -180 ry 0 rz 160 deg; joints [-1.427, 67.216, -10.641, -158.071, 58.523, 168.128]
  Call Extruder(1508.24131)
  MoveL 5313 to (526.53, 440.19, 92) mm, rotated rx 180 ry 0 rz 160 deg; joints [-1.307, 67.592, -11.432, -157.836, 58.163, 167.873]
  Call Extruder(1515.58163)
  MoveL 5314 to (528.65, 441.17, 92) mm, rotated rx 180 ry 0 rz 160 deg; joints [-1.183, 67.952, -12.188, -157.6, 57.823, 167.62]
  Set speed (18.0 mm/s)
  Call Extruder(1523.20857)
  MoveL 5315 to (530.81, 442.28, 92) mm, rotated rx 180 ry 0 rz 160 deg; joints [-1.046, 68.323, -12.966, -157.342, 57.477, 167.35]
  Set speed (18.0 mm/s)
  Call Extruder(1530.92616)
  MoveL 5316 to (532.96, 443.48, 92) mm, rotated rx -180 ry 0 rz 160 deg; joints [-0.899, 68.697, -13.748, -157.07, 57.133, 167.07]
  Set speed (18.0 mm/s)
  Call Extruder(1538.34323)
  MoveL 5317 to (534.98, 444.71, 92) mm, rotated rx 180 ry 0 rz 160 deg; joints [-0.75, 69.053, -14.493, -156.798, 56.81, 166.795]
  Set speed (18.0 mm/s)
  Call Extruder(1546.04475)
  MoveL 5318 to (537.03, 446.06, 92) mm, rotated rx 180 ry 0 rz 160 deg; joints [-0.588, 69.42, -15.258, -156.506, 56.482, 166.502]
  Set speed (18.0 mm/s)
  Call Extruder(1553.51347)
  MoveL 5319 to (538.97, 447.44, 92) mm, rotated rx 180 ry 0 rz 160 deg; joints [-0.423, 69.772, -15.99, -156.212, 56.172, 166.212]
  Call Extruder(1560.97757)
  MoveL 5320 to (540.85, 448.89, 92) mm, rotated rx -180 ry 0 rz 160 deg; joints [-0.252, 70.119, -16.711, -155.909, 55.872, 165.917]
  Call Extruder(1568.61854)
  MoveL 5321 to (542.73, 450.45, 92) mm, rotated rx -180 ry 0 rz 160 deg; joints [-0.07, 70.47, -17.438, -155.59, 55.574, 165.61]
  Call Extruder(0.00000)
  Set speed (18.0 mm/s)
  Call Extruder(7.64948)
  MoveL 5322 to (544.54, 452.07, 92) mm, rotated rx 180 ry 0 rz 160 deg; joints [0.12, 70.815, -18.152, -155.262, 55.285, 165.297]
  Set speed (18.0 mm/s)
  Call Extruder(15.07208)
  MoveL 5323 to (546.25, 453.71, 92) mm, rotated rx 180 ry 0 rz 160 deg; joints [0.309, 71.144, -18.831, -154.936, 55.016, 164.99]
  Set speed (18.0 mm/s)
  Call Extruder(19.29736)
  MoveL 5324 to (547.19, 454.68, 92) mm, rotated rx 180 ry 0 rz 160 deg; joints [0.419, 71.328, -19.212, -154.748, 54.867, 164.814]
  Set speed (18.0 mm/s)
  Call Extruder(23.46807)
  MoveL 5325 to (548.1, 455.64, 92) mm, rotated rx -180 ry 0 rz 160 deg; joints [0.53, 71.508, -19.582, -154.559, 54.724, 164.638]
  Call Extruder(27.69325)
  MoveL 5326 to (549, 456.64, 92) mm, rotated rx -180 ry 0 rz 160 deg; joints [0.644, 71.688, -19.952, -154.367, 54.582, 164.46]
  Set speed (18.0 mm/s)
  Call Extruder(31.87124)
  MoveL 5327 to (549.88, 457.65, 92) mm, rotated rx 180 ry 0 rz 160 deg; joints [0.758, 71.863, -20.313, -154.174, 54.446, 164.282]
  Call Extruder(36.05449)
  MoveL 5328 to (550.73, 458.67, 92) mm, rotated rx 180 ry 0 rz 160 deg; joints [0.874, 72.036, -20.668, -153.979, 54.314, 164.104]
  Set speed (18.0 mm/s)
  Call Extruder(40.30458)
  MoveL 5329 to (551.57, 459.73, 92) mm, rotated rx 180 ry 0 rz 160 deg; joints [0.994, 72.209, -21.024, -153.78, 54.183, 163.922]
  Call Extruder(44.43860)
  MoveL 5330 to (552.37, 460.78, 92) mm, rotated rx 180 ry 0 rz 160 deg; joints [1.112, 72.374, -21.364, -153.584, 54.059, 163.745]
  Set speed (18.0 mm/s)
  Call Extruder(48.76906)
  MoveL 5331 to (553.19, 461.89, 92) mm, rotated rx 180 ry 0 rz 160 deg; joints [1.237, 72.545, -21.715, -153.377, 53.933, 163.559]
  Set speed (18.0 mm/s)
  Call Extruder(52.85321)
  MoveL 5332 to (553.94, 462.96, 92) mm, rotated rx -180 ry 0 rz 160 deg; joints [1.356, 72.703, -22.038, -153.181, 53.819, 163.383]
  Set speed (18.0 mm/s)
  Call Extruder(57.13112)
  MoveL 5333 to (554.69, 464.09, 92) mm, rotated rx -180 ry 0 rz 160 deg; joints [1.483, 72.865, -22.37, -152.974, 53.704, 163.198]
  Set speed (18.0 mm/s)
  Call Extruder(61.23465)
  MoveL 5334 to (555.4, 465.19, 92) mm, rotated rx 180 ry 0 rz 160 deg; joints [1.606, 73.017, -22.683, -152.775, 53.598, 163.022]
  Set speed (18.0 mm/s)
  Call Extruder(65.54246)
  MoveL 5335 to (556.12, 466.36, 92) mm, rotated rx 180 ry 0 rz 160 deg; joints [1.736, 73.174, -23.004, -152.565, 53.49, 162.836]
  Set speed (18.0 mm/s)
  Call Extruder(69.64244)
  MoveL 5336 to (556.78, 467.48, 92) mm, rotated rx 180 ry 0 rz 160 deg; joints [1.861, 73.321, -23.303, -152.364, 53.392, 162.659]
  Set speed (18.0 mm/s)
  Call Extruder(73.85327)
  MoveL 5337 to (557.43, 468.66, 92) mm, rotated rx -180 ry 0 rz 160 deg; joints [1.991, 73.467, -23.602, -152.156, 53.295, 162.479]
  Call Extruder(78.05686)
  MoveL 5338 to (558.06, 469.84, 92) mm, rotated rx -180 ry 0 rz 160 deg; joints [2.122, 73.609, -23.893, -151.949, 53.204, 162.299]
  Set speed (18.0 mm/s)
  Call Extruder(82.24176)
  MoveL 5339 to (558.67, 471.03, 92) mm, rotated rx -180 ry 0 rz 160 deg; joints [2.253, 73.748, -24.176, -151.741, 53.117, 162.12]
  Set speed (18.0 mm/s)
  Call Extruder(86.46760)
  MoveL 5340 to (559.25, 472.24, 92) mm, rotated rx -180 ry 0 rz 160 deg; joints [2.387, 73.883, -24.452, -151.532, 53.034, 161.94]
  Set speed (18.0 mm/s)
  Call Extruder(90.64750)
  MoveL 5341 to (559.8, 473.45, 92) mm, rotated rx -180 ry 0 rz 160 deg; joints [2.52, 74.014, -24.718, -151.324, 52.957, 161.764]
  Set speed (18.0 mm/s)
  Call Extruder(94.96874)
  MoveL 5342 to (560.34, 474.72, 92) mm, rotated rx -180 ry 0 rz 160 deg; joints [2.66, 74.143, -24.981, -151.109, 52.883, 161.583]
  Set speed (18.0 mm/s)
  Call Extruder(99.26146)
  MoveL 5343 to (560.86, 475.98, 92) mm, rotated rx 180 ry 0 rz 160 deg; joints [2.798, 74.27, -25.24, -150.896, 52.812, 161.403]
  Call Extruder(103.35681)
  MoveL 5344 to (561.32, 477.2, 92) mm, rotated rx -180 ry 0 rz 160 deg; joints [2.932, 74.384, -25.472, -150.693, 52.751, 161.234]
  Set speed (18.0 mm/s)
  Call Extruder(107.67147)
  MoveL 5345 to (561.79, 478.49, 92) mm, rotated rx 180 ry 0 rz 160 deg; joints [3.074, 74.503, -25.713, -150.479, 52.691, 161.057]
  Call Extruder(111.76984)
  MoveL 5346 to (562.2, 479.73, 92) mm, rotated rx 180 ry 0 rz 160 deg; joints [3.21, 74.608, -25.928, -150.276, 52.64, 160.891]
  Call Extruder(115.89829)
  MoveL 5347 to (562.6, 480.98, 92) mm, rotated rx 180 ry 0 rz 160 deg; joints [3.347, 74.713, -26.141, -150.072, 52.591, 160.724]
  Set speed (18.0 mm/s)
  Call Extruder(120.19517)
  MoveL 5348 to (562.98, 482.29, 92) mm, rotated rx -180 ry 0 rz 160 deg; joints [3.491, 74.815, -26.348, -149.861, 52.548, 160.554]
  Call Extruder(124.38387)
  MoveL 5349 to (563.34, 483.58, 92) mm, rotated rx -180 ry 0 rz 160 deg; joints [3.631, 74.912, -26.546, -149.655, 52.508, 160.389]
  Set speed (18.0 mm/s)
  Call Extruder(132.70683)
  MoveL 5350 to (563.95, 486.16, 92) mm, rotated rx -180 ry 0 rz 160 deg; joints [3.914, 75.088, -26.903, -149.249, 52.447, 160.068]
  Set speed (18.0 mm/s)
  Call Extruder(141.17099)
  MoveL 5351 to (564.47, 488.8, 92) mm, rotated rx -180 ry 0 rz 160 deg; joints [4.203, 75.248, -27.227, -148.841, 52.406, 159.752]
  Call Extruder(149.56144)
  MoveL 5352 to (564.87, 491.44, 92) mm, rotated rx -180 ry 0 rz 160 deg; joints [4.493, 75.386, -27.506, -148.442, 52.386, 159.451]
  Set speed (18.0 mm/s)
  Call Extruder(158.06631)
  MoveL 5353 to (565.17, 494.14, 92) mm, rotated rx 180 ry 0 rz 160 deg; joints [4.788, 75.504, -27.746, -148.044, 52.387, 159.157]
  Set speed (18.0 mm/s)
  Call Extruder(166.37133)
  MoveL 5354 to (565.35, 496.78, 92) mm, rotated rx -180 ry 0 rz 160 deg; joints [5.078, 75.599, -27.938, -147.662, 52.409, 158.883]
  Set speed (18.0 mm/s)
  Call Extruder(174.76333)
  MoveL 5355 to (565.43, 499.45, 92) mm, rotated rx -180 ry 0 rz 160 deg; joints [5.373, 75.673, -28.088, -147.285, 52.452, 158.621]
  Set speed (18.0 mm/s)
  Call Extruder(183.05993)
  MoveL 5356 to (565.39, 502.09, 92) mm, rotated rx 180 ry 0 rz 160 deg; joints [5.664, 75.724, -28.192, -146.92, 52.514, 158.376]
  Set speed (18.0 mm/s)
  Call Extruder(191.57088)
  MoveL 5357 to (565.26, 504.8, 92) mm, rotated rx 180 ry 0 rz 160 deg; joints [5.964, 75.756, -28.256, -146.556, 52.598, 158.14]
  Set speed (18.0 mm/s)
  Call Extruder(199.88475)
  MoveL 5358 to (565.01, 507.44, 92) mm, rotated rx 180 ry 0 rz 160 deg; joints [6.258, 75.764, -28.271, -146.21, 52.702, 157.927]
  Set speed (18.0 mm/s)
  Call Extruder(208.19716)
  MoveL 5359 to (564.65, 510.07, 92) mm, rotated rx -180 ry 0 rz 160 deg; joints [6.551, 75.75, -28.243, -145.875, 52.824, 157.73]
  Set speed (18.0 mm/s)
  Call Extruder(216.74178)
  MoveL 5360 to (564.18, 512.75, 92) mm, rotated rx 180 ry 0 rz 160 deg; joints [6.853, 75.713, -28.169, -145.542, 52.97, 157.547]
  Set speed (18.0 mm/s)
  Call Extruder(225.20593)
  MoveL 5361 to (563.6, 515.38, 92) mm, rotated rx 180 ry 0 rz 160 deg; joints [7.15, 75.654, -28.05, -145.223, 53.134, 157.383]
  Set speed (18.0 mm/s)
  Call Extruder(229.38259)
  MoveL 5362 to (563.27, 516.67, 92) mm, rotated rx -180 ry 0 rz 160 deg; joints [7.297, 75.615, -27.971, -145.072, 53.222, 157.31]
  Set speed (18.0 mm/s)
  Call Extruder(233.64841)
  MoveL 5363 to (562.91, 517.98, 92) mm, rotated rx -180 ry 0 rz 160 deg; joints [7.446, 75.573, -27.886, -144.918, 53.316, 157.238]
  Set speed (18.0 mm/s)
  Call Extruder(241.79723)
  MoveL 5364 to (562.15, 520.46, 92) mm, rotated rx 180 ry 0 rz 160 deg; joints [7.73, 75.474, -27.685, -144.636, 53.509, 157.117]
  Set speed (18.0 mm/s)
  Call Extruder(246.18425)
  MoveL 5365 to (561.69, 521.78, 92) mm, rotated rx 180 ry 0 rz 160 deg; joints [7.882, 75.411, -27.557, -144.489, 53.621, 157.06]
  Call Extruder(250.26211)
  MoveL 5366 to (561.25, 523, 92) mm, rotated rx 180 ry 0 rz 160 deg; joints [8.023, 75.35, -27.434, -144.355, 53.727, 157.01]
  Set speed (17.9 mm/s)
  Call Extruder(254.59840)
  MoveL 5367 to (560.75, 524.29, 92) mm, rotated rx 180 ry 0 rz 160 deg; joints [8.172, 75.278, -27.287, -144.216, 53.846, 156.963]
  Call Extruder(258.76356)
  MoveL 5368 to (560.25, 525.51, 92) mm, rotated rx 180 ry 0 rz 160 deg; joints [8.315, 75.205, -27.14, -144.085, 53.962, 156.921]
  Set speed (18.0 mm/s)
  Call Extruder(263.00826)
  MoveL 5369 to (559.71, 526.75, 92) mm, rotated rx -180 ry 0 rz 160 deg; joints [8.46, 75.124, -26.975, -143.956, 54.086, 156.885]
  Set speed (18.0 mm/s)
  Call Extruder(267.11834)
  MoveL 5370 to (559.16, 527.94, 92) mm, rotated rx 180 ry 0 rz 160 deg; joints [8.6, 75.043, -26.81, -143.833, 54.209, 156.852]
  Set speed (18.0 mm/s)
  Call Extruder(271.32176)
  MoveL 5371 to (558.58, 529.15, 92) mm, rotated rx -180 ry 0 rz 160 deg; joints [8.743, 74.953, -26.629, -143.71, 54.339, 156.825]
  Set speed (18.0 mm/s)
  Call Extruder(277.78869)
  MoveL 5372 to (557.64, 530.98, 92) mm, rotated rx -180 ry 0 rz 160 deg; joints [8.962, 74.808, -26.333, -143.527, 54.546, 156.791]
  Set speed (18.0 mm/s)
  Call Extruder(283.92118)
  MoveL 5373 to (556.68, 532.69, 92) mm, rotated rx -180 ry 0 rz 160 deg; joints [9.167, 74.657, -26.027, -143.362, 54.752, 156.771]
  Set speed (18.0 mm/s)
  Call Extruder(288.93440)
  MoveL 5374 to (555.87, 534.06, 92) mm, rotated rx 180 ry 0 rz 160 deg; joints [9.333, 74.528, -25.765, -143.231, 54.924, 156.761]
  Call Extruder(292.42134)
  MoveL 5375 to (555.28, 535, 92) mm, rotated rx -180 ry 0 rz 160 deg; joints [9.448, 74.434, -25.573, -143.143, 55.048, 156.758]
  Set speed (18.0 mm/s)
  Call Extruder(296.49345)
  MoveL 5376 to (554.58, 536.1, 92) mm, rotated rx -180 ry 0 rz 160 deg; joints [9.581, 74.321, -25.343, -143.042, 55.194, 156.758]
  Set speed (18.0 mm/s)
  Call Extruder(300.79066)
  MoveL 5377 to (553.81, 537.23, 92) mm, rotated rx 180 ry 0 rz 160 deg; joints [9.721, 74.197, -25.091, -142.939, 55.351, 156.763]
  Call Extruder(304.92781)
  MoveL 5378 to (553.04, 538.31, 92) mm, rotated rx 180 ry 0 rz 160 deg; joints [9.855, 74.073, -24.839, -142.844, 55.507, 156.772]
  Set speed (18.0 mm/s)
  Call Extruder(309.15017)
  MoveL 5379 to (552.25, 539.39, 92) mm, rotated rx 180 ry 0 rz 160 deg; joints [9.99, 73.944, -24.575, -142.749, 55.667, 156.786]
  Set speed (18.0 mm/s)
  Call Extruder(313.38375)
  MoveL 5380 to (551.42, 540.46, 92) mm, rotated rx -180 ry 0 rz 160 deg; joints [10.125, 73.81, -24.301, -142.656, 55.831, 156.804]
  Set speed (18.0 mm/s)
  Call Extruder(317.59857)
  MoveL 5381 to (550.58, 541.5, 92) mm, rotated rx -180 ry 0 rz 160 deg; joints [10.258, 73.672, -24.02, -142.568, 55.997, 156.826]
  Set speed (18.0 mm/s)
  Call Extruder(321.70625)
  MoveL 5382 to (549.74, 542.51, 92) mm, rotated rx 180 ry 0 rz 160 deg; joints [10.386, 73.534, -23.74, -142.484, 56.162, 156.851]
  Call Extruder(325.92616)
  MoveL 5383 to (548.86, 543.52, 92) mm, rotated rx 180 ry 0 rz 160 deg; joints [10.517, 73.389, -23.442, -142.401, 56.333, 156.883]
  Set speed (18.0 mm/s)
  Call Extruder(330.25836)
  MoveL 5384 to (547.93, 544.54, 92) mm, rotated rx 180 ry 0 rz 160 deg; joints [10.65, 73.236, -23.13, -142.319, 56.512, 156.918]
  Set speed (18.0 mm/s)
  Call Extruder(334.36810)
  MoveL 5385 to (547.03, 545.49, 92) mm, rotated rx 180 ry 0 rz 160 deg; joints [10.775, 73.088, -22.827, -142.244, 56.683, 156.956]
  Set speed (18.0 mm/s)
  Call Extruder(338.50452)
  MoveL 5386 to (546.1, 546.43, 92) mm, rotated rx -180 ry 0 rz 160 deg; joints [10.899, 72.935, -22.515, -142.172, 56.858, 156.998]
  Call Extruder(342.77008)
  MoveL 5387 to (545.13, 547.38, 92) mm, rotated rx 180 ry 0 rz 160 deg; joints [11.026, 72.775, -22.185, -142.1, 57.041, 157.046]
  Call Extruder(346.89968)
  MoveL 5388 to (544.17, 548.28, 92) mm, rotated rx -180 ry 0 rz 160 deg; joints [11.147, 72.617, -21.861, -142.032, 57.219, 157.095]
  Call Extruder(351.17120)
  MoveL 5389 to (543.15, 549.18, 92) mm, rotated rx 180 ry 0 rz 160 deg; joints [11.271, 72.45, -21.519, -141.966, 57.405, 157.15]
  Set speed (18.0 mm/s)
  Call Extruder(355.31232)
  MoveL 5390 to (542.15, 550.04, 92) mm, rotated rx 180 ry 0 rz 160 deg; joints [11.39, 72.285, -21.181, -141.904, 57.588, 157.207]
  Set speed (18.0 mm/s)
  Call Extruder(359.50165)
  MoveL 5391 to (541.12, 550.89, 92) mm, rotated rx -180 ry 0 rz 160 deg; joints [11.509, 72.116, -20.833, -141.845, 57.774, 157.268]
  Set speed (18.0 mm/s)
  Call Extruder(363.77471)
  MoveL 5392 to (540.05, 551.74, 92) mm, rotated rx 180 ry 0 rz 160 deg; joints [11.628, 71.94, -20.473, -141.786, 57.966, 157.334]
  Call Extruder(367.90945)
  MoveL 5393 to (539, 552.53, 92) mm, rotated rx -180 ry 0 rz 160 deg; joints [11.742, 71.768, -20.118, -141.733, 58.153, 157.402]
  Set speed (18.0 mm/s)
  Call Extruder(372.18199)
  MoveL 5394 to (537.9, 553.33, 92) mm, rotated rx 180 ry 0 rz 160 deg; joints [11.858, 71.587, -19.746, -141.681, 58.347, 157.475]
  Set speed (18.0 mm/s)
  Call Extruder(376.35900)
  MoveL 5395 to (536.81, 554.09, 92) mm, rotated rx 180 ry 0 rz 160 deg; joints [11.969, 71.409, -19.377, -141.632, 58.539, 157.55]
  Set speed (18.0 mm/s)
  Call Extruder(380.50383)
  MoveL 5396 to (535.71, 554.83, 92) mm, rotated rx -180 ry 0 rz 160 deg; joints [12.079, 71.229, -19.007, -141.586, 58.73, 157.627]
  Set speed (18.0 mm/s)
  Call Extruder(384.71833)
  MoveL 5397 to (534.58, 555.55, 92) mm, rotated rx 180 ry 0 rz 160 deg; joints [12.188, 71.044, -18.625, -141.542, 58.926, 157.709]
  Call Extruder(388.92068)
  MoveL 5398 to (533.43, 556.24, 92) mm, rotated rx 180 ry 0 rz 160 deg; joints [12.294, 70.858, -18.24, -141.501, 59.122, 157.794]
  Set speed (18.0 mm/s)
  Call Extruder(393.11888)
  MoveL 5399 to (532.28, 556.91, 92) mm, rotated rx 180 ry 0 rz 160 deg; joints [12.399, 70.669, -17.851, -141.462, 59.319, 157.882]
  Set speed (18.0 mm/s)
  Call Extruder(397.43166)
  MoveL 5400 to (531.08, 557.58, 92) mm, rotated rx 180 ry 0 rz 160 deg; joints [12.505, 70.474, -17.447, -141.425, 59.522, 157.975]
  Set speed (18.0 mm/s)
  Call Extruder(403.56967)
  MoveL 5401 to (529.34, 558.49, 92) mm, rotated rx 180 ry 0 rz 160 deg; joints [12.652, 70.193, -16.864, -141.377, 59.812, 158.113]
  Set speed (18.0 mm/s)
  Call Extruder(409.82225)
  MoveL 5402 to (527.54, 559.35, 92) mm, rotated rx 180 ry 0 rz 160 deg; joints [12.798, 69.903, -16.262, -141.334, 60.11, 158.26]
  Set speed (18.0 mm/s)
  Call Extruder(414.20296)
  MoveL 5403 to (526.27, 559.92, 92) mm, rotated rx 180 ry 0 rz 160 deg; joints [12.896, 69.698, -15.835, -141.308, 60.319, 158.367]
  Set speed (18.0 mm/s)
  Call Extruder(418.53691)
  MoveL 5404 to (525, 560.47, 92) mm, rotated rx -180 ry 0 rz 160 deg; joints [12.992, 69.494, -15.412, -141.284, 60.526, 158.475]
  Set speed (18.0 mm/s)
  Call Extruder(426.66164)
  MoveL 5405 to (522.59, 561.41, 92) mm, rotated rx 180 ry 0 rz 160 deg; joints [13.164, 69.108, -14.607, -141.246, 60.916, 158.685]
  Set speed (18.0 mm/s)
  Call Extruder(431.03573)
  MoveL 5406 to (521.28, 561.87, 92) mm, rotated rx -180 ry 0 rz 160 deg; joints [13.253, 68.898, -14.169, -141.231, 61.126, 158.803]
  Set speed (18.0 mm/s)
  Call Extruder(435.15086)
  MoveL 5407 to (520.04, 562.29, 92) mm, rotated rx 180 ry 0 rz 160 deg; joints [13.335, 68.701, -13.757, -141.218, 61.323, 158.914]
  Set speed (18.0 mm/s)
  Call Extruder(439.38186)
  MoveL 5408 to (518.75, 562.68, 92) mm, rotated rx -180 ry 0 rz 160 deg; joints [13.416, 68.496, -13.328, -141.208, 61.526, 159.032]
  Set speed (18.0 mm/s)
  Call Extruder(443.46431)
  MoveL 5409 to (517.5, 563.04, 92) mm, rotated rx -180 ry 0 rz 160 deg; joints [13.493, 68.298, -12.915, -141.199, 61.722, 159.147]
  Set speed (17.9 mm/s)
  Call Extruder(447.27726)
  MoveL 5410 to (516.33, 563.36, 92) mm, rotated rx 180 ry 0 rz 160 deg; joints [13.562, 68.113, -12.526, -141.195, 61.905, 159.257]
  Set speed (17.9 mm/s)
  Call Extruder(451.88750)
  MoveL 5411 to (514.91, 563.71, 92) mm, rotated rx -180 ry 0 rz 160 deg; joints [13.643, 67.888, -12.055, -141.191, 62.125, 159.392]
  Set speed (18.0 mm/s)
  Call Extruder(460.41528)
  MoveL 5412 to (512.25, 564.27, 92) mm, rotated rx 180 ry 0 rz 160 deg; joints [13.785, 67.47, -11.176, -141.192, 62.534, 159.648]
  Call Extruder(468.88158)
  MoveL 5413 to (509.59, 564.72, 92) mm, rotated rx 180 ry 0 rz 160 deg; joints [13.914, 67.054, -10.299, -141.204, 62.938, 159.91]
  Set speed (18.0 mm/s)
  Call Extruder(477.19101)
  MoveL 5414 to (506.96, 565.06, 92) mm, rotated rx -180 ry 0 rz 160 deg; joints [14.031, 66.644, -9.434, -141.225, 63.333, 160.175]
  Call Extruder(485.63746)
  MoveL 5415 to (504.28, 565.29, 92) mm, rotated rx 180 ry 0 rz 160 deg; joints [14.138, 66.228, -8.553, -141.258, 63.731, 160.45]
  Set speed (18.0 mm/s)
  Call Extruder(494.08769)
  MoveL 5416 to (501.59, 565.41, 92) mm, rotated rx 180 ry 0 rz 160 deg; joints [14.233, 65.812, -7.67, -141.301, 64.127, 160.731]
  Call Extruder(502.31935)
  MoveL 5417 to (498.97, 565.42, 92) mm, rotated rx 180 ry 0 rz 160 deg; joints [14.315, 65.408, -6.81, -141.352, 64.51, 161.01]
  Set speed (10.0 mm/s)
  MoveL 5418 to (498.97, 565.42, 96) mm, rotated rx 180 ry 0 rz 160 deg; joints [14.315, 64.766, -6.499, -141.253, 64.252, 160.781]
  Set speed (120.0 mm/s)
  MoveL 5419 to (498.97, 565.46, 96) mm, rotated rx 180 ry 0 rz 160 deg; joints [14.319, 64.768, -6.504, -141.248, 64.251, 160.777]
  Set speed (18.0 mm/s)
  Call Extruder(510.87808)
  MoveL 5420 to (496.25, 565.36, 96) mm, rotated rx 180 ry 0 rz 160 deg; joints [14.391, 64.348, -5.613, -141.314, 64.642, 161.071]
  Set speed (18.0 mm/s)
  Call Extruder(519.30131)
  MoveL 5421 to (493.57, 565.15, 96) mm, rotated rx 180 ry 0 rz 160 deg; joints [14.449, 63.938, -4.739, -141.389, 65.022, 161.365]
  Set speed (18.0 mm/s)
  Call Extruder(527.64022)
  MoveL 5422 to (490.93, 564.83, 96) mm, rotated rx 180 ry 0 rz 160 deg; joints [14.493, 63.534, -3.878, -141.474, 65.394, 161.659]
  Set speed (18.0 mm/s)
  Call Extruder(535.93924)
  MoveL 5423 to (488.32, 564.41, 96) mm, rotated rx -180 ry 0 rz 160 deg; joints [14.525, 63.135, -3.025, -141.57, 65.759, 161.956]
  Set speed (18.0 mm/s)
  Call Extruder(544.52961)
  MoveL 5424 to (485.63, 563.87, 96) mm, rotated rx 180 ry 0 rz 160 deg; joints [14.543, 62.726, -2.149, -141.68, 66.131, 162.266]
  Set speed (18.0 mm/s)
  Call Extruder(548.70039)
  MoveL 5425 to (484.34, 563.56, 96) mm, rotated rx 180 ry 0 rz 160 deg; joints [14.546, 62.529, -1.727, -141.738, 66.309, 162.417]
  Set speed (18.0 mm/s)
  Call Extruder(552.72403)
  MoveL 5426 to (483.1, 563.25, 96) mm, rotated rx -180 ry 0 rz 160 deg; joints [14.547, 62.341, -1.322, -141.795, 66.48, 162.563]
  Call Extruder(557.09212)
  MoveL 5427 to (481.77, 562.87, 96) mm, rotated rx 180 ry 0 rz 160 deg; joints [14.543, 62.138, -0.884, -141.862, 66.663, 162.723]
  Call Extruder(561.36196)
  MoveL 5428 to (480.46, 562.48, 96) mm, rotated rx 180 ry 0 rz 160 deg; joints [14.537, 61.941, -0.459, -141.929, 66.841, 162.878]
  Call Extruder(565.46927)
  MoveL 5429 to (479.22, 562.07, 96) mm, rotated rx 180 ry 0 rz 160 deg; joints [14.526, 61.752, -0.052, -141.998, 67.009, 163.029]
  Set speed (18.0 mm/s)
  Call Extruder(569.54903)
  MoveL 5430 to (477.99, 561.65, 96) mm, rotated rx 180 ry 0 rz 160 deg; joints [14.514, 61.567, 0.35, -142.067, 67.176, 163.178]
  Set speed (18.0 mm/s)
  Call Extruder(573.93524)
  MoveL 5431 to (476.68, 561.17, 96) mm, rotated rx -180 ry 0 rz 160 deg; joints [14.495, 61.369, 0.779, -142.146, 67.353, 163.34]
  Set speed (18.0 mm/s)
  Call Extruder(578.14041)
  MoveL 5432 to (475.44, 560.68, 96) mm, rotated rx -180 ry 0 rz 160 deg; joints [14.475, 61.18, 1.187, -142.223, 67.521, 163.494]
  Set speed (18.0 mm/s)
  Call Extruder(582.75003)
  MoveL 5433 to (474.09, 560.11, 96) mm, rotated rx 180 ry 0 rz 160 deg; joints [14.447, 60.976, 1.632, -142.313, 67.703, 163.664]
  Set speed (18.0 mm/s)
  Call Extruder(586.49839)
  MoveL 5434 to (472.99, 559.63, 96) mm, rotated rx -180 ry 0 rz 160 deg; joints [14.422, 60.811, 1.991, -142.387, 67.849, 163.801]
  Set speed (18.0 mm/s)
  Call Extruder(590.63013)
  MoveL 5435 to (471.8, 559.08, 96) mm, rotated rx -180 ry 0 rz 160 deg; joints [14.39, 60.63, 2.383, -142.472, 68.009, 163.954]
  Set speed (18.0 mm/s)
  Call Extruder(594.88275)
  MoveL 5436 to (470.58, 558.48, 96) mm, rotated rx -180 ry 0 rz 160 deg; joints [14.354, 60.447, 2.784, -142.563, 68.171, 164.11]
  Set speed (18.0 mm/s)
  Call Extruder(598.06081)
  MoveL 5437 to (469.68, 558.02, 96) mm, rotated rx -180 ry 0 rz 160 deg; joints [14.324, 60.311, 3.081, -142.633, 68.291, 164.227]
  Set speed (18.0 mm/s)
  Call Extruder(603.24082)
  MoveL 5438 to (468.23, 557.24, 96) mm, rotated rx 180 ry 0 rz 160 deg; joints [14.271, 60.091, 3.561, -142.751, 68.484, 164.417]
  Set speed (18.0 mm/s)
  Call Extruder(607.48064)
  MoveL 5439 to (467.05, 556.57, 96) mm, rotated rx -180 ry 0 rz 160 deg; joints [14.223, 59.914, 3.95, -142.851, 68.64, 164.573]
  Set speed (18.0 mm/s)
  Call Extruder(611.75711)
  MoveL 5440 to (465.88, 555.87, 96) mm, rotated rx 180 ry 0 rz 160 deg; joints [14.171, 59.737, 4.338, -142.954, 68.794, 164.729]
  Call Extruder(615.90462)
  MoveL 5441 to (464.76, 555.17, 96) mm, rotated rx -180 ry 0 rz 160 deg; joints [14.116, 59.567, 4.711, -143.057, 68.942, 164.88]
  Set speed (18.0 mm/s)
  Call Extruder(620.24894)
  MoveL 5442 to (463.6, 554.41, 96) mm, rotated rx 180 ry 0 rz 160 deg; joints [14.056, 59.392, 5.097, -143.169, 69.095, 165.038]
  Call Extruder(624.29237)
  MoveL 5443 to (462.54, 553.68, 96) mm, rotated rx -180 ry 0 rz 160 deg; joints [13.995, 59.231, 5.452, -143.275, 69.235, 165.184]
  Set speed (18.0 mm/s)
  Call Extruder(628.49077)
  MoveL 5444 to (461.45, 552.91, 96) mm, rotated rx 180 ry 0 rz 160 deg; joints [13.929, 59.066, 5.816, -143.389, 69.377, 165.336]
  Set speed (18.0 mm/s)
  Call Extruder(632.66278)
  MoveL 5445 to (460.38, 552.11, 96) mm, rotated rx -180 ry 0 rz 160 deg; joints [13.859, 58.904, 6.174, -143.505, 69.517, 165.486]
  Set speed (18.0 mm/s)
  Call Extruder(636.82880)
  MoveL 5446 to (459.33, 551.3, 96) mm, rotated rx -180 ry 0 rz 160 deg; joints [13.786, 58.745, 6.526, -143.623, 69.654, 165.635]
  Call Extruder(641.07329)
  MoveL 5447 to (458.28, 550.45, 96) mm, rotated rx 180 ry 0 rz 160 deg; joints [13.707, 58.585, 6.88, -143.748, 69.792, 165.786]
  Call Extruder(645.27693)
  MoveL 5448 to (457.25, 549.58, 96) mm, rotated rx 180 ry 0 rz 160 deg; joints [13.625, 58.429, 7.226, -143.873, 69.925, 165.934]
  Set speed (18.0 mm/s)
  Call Extruder(649.42667)
  MoveL 5449 to (456.26, 548.71, 96) mm, rotated rx -180 ry 0 rz 160 deg; joints [13.541, 58.278, 7.562, -144, 70.054, 166.08]
  Set speed (18.0 mm/s)
  Call Extruder(653.68568)
  MoveL 5450 to (455.26, 547.79, 96) mm, rotated rx 180 ry 0 rz 160 deg; joints [13.45, 58.126, 7.902, -144.134, 70.184, 166.229]
  Set speed (18.0 mm/s)
  Call Extruder(657.82977)
  MoveL 5451 to (454.31, 546.88, 96) mm, rotated rx 180 ry 0 rz 160 deg; joints [13.358, 57.98, 8.228, -144.266, 70.308, 166.372]
  Call Extruder(662.05267)
  MoveL 5452 to (453.35, 545.93, 96) mm, rotated rx 180 ry 0 rz 160 deg; joints [13.261, 57.833, 8.554, -144.404, 70.432, 166.518]
  Set speed (18.0 mm/s)
  Call Extruder(666.22126)
  MoveL 5453 to (452.43, 544.97, 96) mm, rotated rx 180 ry 0 rz 160 deg; joints [13.161, 57.692, 8.871, -144.543, 70.551, 166.66]
  Set speed (18.0 mm/s)
  Call Extruder(670.49842)
  MoveL 5454 to (451.5, 543.97, 96) mm, rotated rx -180 ry 0 rz 160 deg; joints [13.054, 57.549, 9.19, -144.689, 70.67, 166.805]
  Set speed (18.0 mm/s)
  Call Extruder(674.61087)
  MoveL 5455 to (450.63, 542.99, 96) mm, rotated rx 180 ry 0 rz 160 deg; joints [12.949, 57.415, 9.491, -144.832, 70.783, 166.943]
  Set speed (18.0 mm/s)
  Call Extruder(678.42177)
  MoveL 5456 to (449.84, 542.07, 96) mm, rotated rx -180 ry 0 rz 160 deg; joints [12.847, 57.293, 9.765, -144.966, 70.884, 167.07]
  Set speed (18.0 mm/s)
  Call Extruder(683.07740)
  MoveL 5457 to (448.9, 540.92, 96) mm, rotated rx 180 ry 0 rz 160 deg; joints [12.72, 57.147, 10.093, -145.134, 71.005, 167.223]
  Set speed (18.0 mm/s)
  Call Extruder(687.27209)
  MoveL 5458 to (448.08, 539.87, 96) mm, rotated rx -180 ry 0 rz 160 deg; joints [12.601, 57.019, 10.382, -145.288, 71.111, 167.36]
  Call Extruder(691.50723)
  MoveL 5459 to (447.27, 538.79, 96) mm, rotated rx -180 ry 0 rz 160 deg; joints [12.477, 56.892, 10.668, -145.446, 71.215, 167.496]
  Set speed (18.0 mm/s)
  Call Extruder(695.68690)
  MoveL 5460 to (446.49, 537.71, 96) mm, rotated rx 180 ry 0 rz 160 deg; joints [12.352, 56.77, 10.944, -145.605, 71.315, 167.63]
  Set speed (18.0 mm/s)
  Call Extruder(699.88365)
  MoveL 5461 to (445.73, 536.61, 96) mm, rotated rx -180 ry 0 rz 160 deg; joints [12.222, 56.65, 11.215, -145.767, 71.412, 167.762]
  Set speed (18.0 mm/s)
  Call Extruder(704.09987)
  MoveL 5462 to (444.99, 535.49, 96) mm, rotated rx 180 ry 0 rz 160 deg; joints [12.089, 56.533, 11.48, -145.933, 71.506, 167.894]
  Set speed (18.0 mm/s)
  Call Extruder(708.36783)
  MoveL 5463 to (444.26, 534.34, 96) mm, rotated rx -180 ry 0 rz 160 deg; joints [11.951, 56.417, 11.742, -146.103, 71.599, 168.025]
  Set speed (18.0 mm/s)
  Call Extruder(712.45815)
  MoveL 5464 to (443.59, 533.22, 96) mm, rotated rx 180 ry 0 rz 160 deg; joints [11.814, 56.31, 11.986, -146.269, 71.684, 168.15]
  Call Extruder(716.78372)
  MoveL 5465 to (442.9, 532.03, 96) mm, rotated rx 180 ry 0 rz 160 deg; joints [11.667, 56.199, 12.237, -146.446, 71.771, 168.279]
  Set speed (18.0 mm/s)
  Call Extruder(720.83645)
  MoveL 5466 to (442.28, 530.89, 96) mm, rotated rx 180 ry 0 rz 160 deg; joints [11.526, 56.099, 12.466, -146.615, 71.85, 168.399]
  Call Extruder(725.08625)
  MoveL 5467 to (441.66, 529.69, 96) mm, rotated rx 180 ry 0 rz 160 deg; joints [11.375, 55.996, 12.699, -146.794, 71.929, 168.523]
  Set speed (18.0 mm/s)
  Call Extruder(729.23603)
  MoveL 5468 to (441.07, 528.51, 96) mm, rotated rx -180 ry 0 rz 160 deg; joints [11.225, 55.9, 12.92, -146.971, 72.003, 168.642]
  Set speed (18.0 mm/s)
  Call Extruder(733.58307)
  MoveL 5469 to (440.48, 527.25, 96) mm, rotated rx 180 ry 0 rz 160 deg; joints [11.063, 55.802, 13.142, -147.159, 72.076, 168.765]
  Set speed (18.0 mm/s)
  Call Extruder(737.78080)
  MoveL 5470 to (439.94, 526.03, 96) mm, rotated rx -180 ry 0 rz 160 deg; joints [10.906, 55.711, 13.351, -147.342, 72.144, 168.882]
  Set speed (18.0 mm/s)
  Call Extruder(745.99851)
  MoveL 5471 to (438.94, 523.61, 96) mm, rotated rx 180 ry 0 rz 160 deg; joints [10.588, 55.542, 13.738, -147.707, 72.267, 169.104]
  Set speed (17.9 mm/s)
  Call Extruder(749.90777)
  MoveL 5472 to (438.51, 522.45, 96) mm, rotated rx 180 ry 0 rz 160 deg; joints [10.433, 55.467, 13.91, -147.884, 72.32, 169.207]
  Call Extruder(754.72951)
  MoveL 5473 to (438, 521, 96) mm, rotated rx 180 ry 0 rz 160 deg; joints [10.24, 55.377, 14.116, -148.103, 72.383, 169.333]
  Set speed (18.0 mm/s)
  Call Extruder(758.81334)
  MoveL 5474 to (437.6, 519.76, 96) mm, rotated rx 180 ry 0 rz 160 deg; joints [10.072, 55.305, 14.281, -148.291, 72.431, 169.436]
  Set speed (18.0 mm/s)
  Call Extruder(762.81761)
  MoveL 5475 to (437.22, 518.55, 96) mm, rotated rx -180 ry 0 rz 160 deg; joints [9.907, 55.237, 14.438, -148.476, 72.477, 169.536]
  Call Extruder(767.23967)
  MoveL 5476 to (436.84, 517.19, 96) mm, rotated rx 180 ry 0 rz 160 deg; joints [9.721, 55.166, 14.6, -148.683, 72.522, 169.644]
  Set speed (18.0 mm/s)
  Call Extruder(771.29199)
  MoveL 5477 to (436.51, 515.95, 96) mm, rotated rx 180 ry 0 rz 160 deg; joints [9.55, 55.104, 14.744, -148.873, 72.561, 169.742]
  Set speed (18.0 mm/s)
  Call Extruder(775.64074)
  MoveL 5478 to (436.19, 514.6, 96) mm, rotated rx 180 ry 0 rz 160 deg; joints [9.363, 55.042, 14.887, -149.079, 72.597, 169.843]
  Set speed (18.0 mm/s)
  Call Extruder(779.82420)
  MoveL 5479 to (435.9, 513.3, 96) mm, rotated rx -180 ry 0 rz 160 deg; joints [9.181, 54.985, 15.019, -149.278, 72.629, 169.939]
  Set speed (18.0 mm/s)
  Call Extruder(788.27755)
  MoveL 5480 to (435.41, 510.65, 96) mm, rotated rx 180 ry 0 rz 160 deg; joints [8.808, 54.881, 15.26, -149.685, 72.682, 170.127]
  Set speed (18.0 mm/s)
  Call Extruder(796.67859)
  MoveL 5481 to (435.02, 508, 96) mm, rotated rx -180 ry 0 rz 160 deg; joints [8.43, 54.791, 15.467, -150.093, 72.719, 170.304]
  Set speed (18.0 mm/s)
  Call Extruder(805.07292)
  MoveL 5482 to (434.75, 505.34, 96) mm, rotated rx 180 ry 0 rz 160 deg; joints [8.047, 54.716, 15.64, -150.504, 72.741, 170.472]
  Set speed (18.0 mm/s)
  Call Extruder(813.31834)
  MoveL 5483 to (434.59, 502.71, 96) mm, rotated rx -180 ry 0 rz 160 deg; joints [7.666, 54.657, 15.777, -150.909, 72.746, 170.629]
  Call Extruder(821.79495)
  MoveL 5484 to (434.53, 500.01, 96) mm, rotated rx 180 ry 0 rz 160 deg; joints [7.271, 54.61, 15.886, -151.327, 72.737, 170.782]
  Call Extruder(829.43957)
  MoveL 5485 to (434.58, 497.58, 96) mm, rotated rx -180 ry 0 rz 160 deg; joints [6.912, 54.581, 15.953, -151.704, 72.713, 170.911]
  Call Extruder(836.84910)
  MoveL 5486 to (434.71, 495.22, 96) mm, rotated rx -180 ry 0 rz 160 deg; joints [6.563, 54.564, 15.992, -152.068, 72.678, 171.03]
  Set speed (18.0 mm/s)
  Call Extruder(844.47208)
  MoveL 5487 to (434.93, 492.8, 96) mm, rotated rx -180 ry 0 rz 160 deg; joints [6.203, 54.559, 16.005, -152.442, 72.629, 171.144]
  Call Extruder(852.04231)
  MoveL 5488 to (435.24, 490.41, 96) mm, rotated rx 180 ry 0 rz 160 deg; joints [5.845, 54.566, 15.99, -152.811, 72.566, 171.251]
  Set speed (18.0 mm/s)
  Call Extruder(859.46030)
  MoveL 5489 to (435.63, 488.08, 96) mm, rotated rx 180 ry 0 rz 160 deg; joints [5.496, 54.583, 15.948, -153.17, 72.492, 171.348]
  Set speed (18.0 mm/s)
  Call Extruder(867.10926)
  MoveL 5490 to (436.12, 485.69, 96) mm, rotated rx -180 ry 0 rz 160 deg; joints [5.137, 54.614, 15.878, -153.536, 72.403, 171.442]
  Set speed (18.0 mm/s)
  Call Extruder(874.72378)
  MoveL 5491 to (436.69, 483.33, 96) mm, rotated rx -180 ry 0 rz 160 deg; joints [4.782, 54.656, 15.78, -153.897, 72.301, 171.528]
  Set speed (18.0 mm/s)
  Call Extruder(882.28539)
  MoveL 5492 to (437.35, 481.01, 96) mm, rotated rx 180 ry 0 rz 160 deg; joints [4.432, 54.709, 15.656, -154.25, 72.186, 171.606]
  Set speed (18.0 mm/s)
  Call Extruder(889.79207)
  MoveL 5493 to (438.09, 478.73, 96) mm, rotated rx 180 ry 0 rz 160 deg; joints [4.089, 54.775, 15.505, -154.595, 72.059, 171.676]
  Call Extruder(897.32609)
  MoveL 5494 to (438.91, 476.48, 96) mm, rotated rx -180 ry 0 rz 160 deg; joints [3.749, 54.851, 15.328, -154.935, 71.919, 171.741]
  Set speed (18.0 mm/s)
  Call Extruder(904.18049)
  MoveL 5495 to (439.73, 474.45, 96) mm, rotated rx 180 ry 0 rz 160 deg; joints [3.444, 54.93, 15.145, -155.238, 71.781, 171.794]
  Set speed (18.0 mm/s)
  Call Extruder(912.62813)
  MoveL 5496 to (440.83, 472, 96) mm, rotated rx -180 ry 0 rz 160 deg; joints [3.075, 55.042, 14.888, -155.603, 71.596, 171.851]
  Set speed (18.0 mm/s)
  Call Extruder(919.96832)
  MoveL 5497 to (441.87, 469.9, 96) mm, rotated rx -180 ry 0 rz 160 deg; joints [2.761, 55.15, 14.639, -155.911, 71.423, 171.894]
  Set speed (18.0 mm/s)
  Call Extruder(927.60432)
  MoveL 5498 to (443.02, 467.76, 96) mm, rotated rx -180 ry 0 rz 160 deg; joints [2.441, 55.273, 14.354, -156.224, 71.231, 171.932]
  Set speed (18.0 mm/s)
  Call Extruder(935.31385)
  MoveL 5499 to (444.27, 465.65, 96) mm, rotated rx -180 ry 0 rz 160 deg; joints [2.125, 55.41, 14.041, -156.529, 71.024, 171.964]
  Set speed (18.0 mm/s)
  Call Extruder(942.79153)
  MoveL 5500 to (445.56, 463.64, 96) mm, rotated rx 180 ry 0 rz 160 deg; joints [1.827, 55.553, 13.712, -156.816, 70.813, 171.988]
  Set speed (18.0 mm/s)
  Call Extruder(950.35097)
  MoveL 5501 to (446.94, 461.66, 96) mm, rotated rx 180 ry 0 rz 160 deg; joints [1.535, 55.709, 13.356, -157.095, 70.587, 172.006]
  Set speed (18.0 mm/s)
  Call Extruder(957.99166)
  MoveL 5502 to (448.4, 459.72, 96) mm, rotated rx 180 ry 0 rz 160 deg; joints [1.249, 55.877, 12.971, -157.366, 70.348, 172.018]
  Call Extruder(965.47773)
  MoveL 5503 to (449.9, 457.86, 96) mm, rotated rx -180 ry 0 rz 160 deg; joints [0.979, 56.053, 12.57, -157.62, 70.103, 172.023]
  Set speed (18.0 mm/s)
  Call Extruder(973.03500)
  MoveL 5504 to (451.49, 456.05, 96) mm, rotated rx 180 ry 0 rz 160 deg; joints [0.715, 56.24, 12.144, -157.864, 69.845, 172.021]
  Call Extruder(980.82663)
  MoveL 5505 to (453.19, 454.24, 96) mm, rotated rx 180 ry 0 rz 160 deg; joints [0.455, 56.444, 11.681, -158.104, 69.569, 172.013]
  Set speed (18.0 mm/s)
  Call Extruder(988.14383)
  MoveL 5506 to (454.85, 452.6, 96) mm, rotated rx 180 ry 0 rz 160 deg; joints [0.221, 56.645, 11.225, -158.316, 69.3, 171.999]
  Call Extruder(995.71182)
  MoveL 5507 to (456.63, 450.97, 96) mm, rotated rx 180 ry 0 rz 160 deg; joints [-0.01, 56.863, 10.733, -158.522, 69.012, 171.978]
  Set speed (18.0 mm/s)
  Call Extruder(1003.35528)
  MoveL 5508 to (458.48, 449.39, 96) mm, rotated rx -180 ry 0 rz 160 deg; joints [-0.232, 57.093, 10.215, -158.717, 68.713, 171.951]
  Set speed (18.0 mm/s)
  Call Extruder(1011.20662)
  MoveL 5509 to (460.44, 447.84, 96) mm, rotated rx -180 ry 0 rz 160 deg; joints [-0.448, 57.339, 9.663, -158.903, 68.396, 171.915]
  Set speed (18.0 mm/s)
  Call Extruder(1018.29975)
  MoveL 5510 to (462.27, 446.5, 96) mm, rotated rx -180 ry 0 rz 160 deg; joints [-0.632, 57.569, 9.146, -159.058, 68.103, 171.877]
  Set speed (18.0 mm/s)
  Call Extruder(1025.96896)
  MoveL 5511 to (464.29, 445.13, 96) mm, rotated rx 180 ry 0 rz 160 deg; joints [-0.819, 57.827, 8.568, -159.211, 67.778, 171.83]
  Set speed (18.0 mm/s)
  Call Extruder(1033.60816)
  MoveL 5512 to (466.35, 443.85, 96) mm, rotated rx 180 ry 0 rz 160 deg; joints [-0.992, 58.093, 7.974, -159.349, 67.447, 171.775]
  Set speed (18.0 mm/s)
  Call Extruder(1041.17946)
  MoveL 5513 to (468.45, 442.64, 96) mm, rotated rx 180 ry 0 rz 160 deg; joints [-1.152, 58.365, 7.368, -159.471, 67.111, 171.714]
  Set speed (18.0 mm/s)
  Call Extruder(1049.60899)
  MoveL 5514 to (470.82, 441.4, 96) mm, rotated rx 180 ry 0 rz 160 deg; joints [-1.315, 58.677, 6.675, -159.591, 66.731, 171.638]
  Set speed (18.0 mm/s)
  Call Extruder(1056.31702)
  MoveL 5515 to (472.75, 440.48, 96) mm, rotated rx 180 ry 0 rz 160 deg; joints [-1.434, 58.933, 6.11, -159.672, 66.423, 171.571]
  Set speed (18.0 mm/s)
  Call Extruder(1063.90064)
  MoveL 5516 to (474.96, 439.51, 96) mm, rotated rx -180 ry 0 rz 160 deg; joints [-1.557, 59.229, 5.456, -159.75, 66.069, 171.489]
  Set speed (18.0 mm/s)
  Call Extruder(1071.30969)
  MoveL 5517 to (477.16, 438.65, 96) mm, rotated rx 180 ry 0 rz 160 deg; joints [-1.665, 59.525, 4.803, -159.812, 65.719, 171.402]
  Set speed (18.0 mm/s)
  Call Extruder(1078.96999)
  MoveL 5518 to (479.46, 437.84, 96) mm, rotated rx 180 ry 0 rz 160 deg; joints [-1.764, 59.839, 4.114, -159.86, 65.351, 171.304]
  Set speed (18.0 mm/s)
  Call Extruder(1086.42794)
  MoveL 5519 to (481.73, 437.14, 96) mm, rotated rx -180 ry 0 rz 160 deg; joints [-1.848, 60.151, 3.43, -159.893, 64.99, 171.202]
  Call Extruder(1094.05279)
  MoveL 5520 to (484.08, 436.5, 96) mm, rotated rx -180 ry 0 rz 160 deg; joints [-1.922, 60.476, 2.719, -159.911, 64.616, 171.09]
  Set speed (18.0 mm/s)
  Call Extruder(1101.70027)
  MoveL 5521 to (486.46, 435.95, 96) mm, rotated rx 180 ry 0 rz 160 deg; joints [-1.984, 60.809, 1.995, -159.914, 64.238, 170.969]
  Call Extruder(1109.11866)
  MoveL 5522 to (488.78, 435.5, 96) mm, rotated rx 180 ry 0 rz 160 deg; joints [-2.032, 61.137, 1.281, -159.903, 63.869, 170.845]
  Set speed (18.0 mm/s)
  Call Extruder(1116.40586)
  MoveL 5523 to (491.07, 435.15, 96) mm, rotated rx -180 ry 0 rz 160 deg; joints [-2.067, 61.464, 0.572, -159.877, 63.504, 170.716]
  Set speed (18.0 mm/s)
  Call Extruder(1124.34802)
  MoveL 5524 to (493.58, 434.85, 96) mm, rotated rx 180 ry 0 rz 160 deg; joints [-2.094, 61.826, -0.21, -159.833, 63.105, 170.567]
  Set speed (18.0 mm/s)
  Call Extruder(1131.86454)
  MoveL 5525 to (495.97, 434.66, 96) mm, rotated rx -180 ry 0 rz 160 deg; joints [-2.107, 62.173, -0.959, -159.777, 62.725, 170.418]
  Set speed (18.0 mm/s)
  Call Extruder(1139.51338)
  MoveL 5526 to (498.41, 434.56, 96) mm, rotated rx 180 ry 0 rz 160 deg; joints [-2.109, 62.531, -1.73, -159.705, 62.338, 170.258]
  Call Extruder(1146.99220)
  MoveL 5527 to (500.79, 434.54, 96) mm, rotated rx -180 ry 0 rz 160 deg; joints [-2.1, 62.885, -2.489, -159.62, 61.959, 170.094]
  Set speed (18.0 mm/s)
  Call Extruder(1154.43172)
  MoveL 5528 to (503.16, 434.61, 96) mm, rotated rx -180 ry 0 rz 160 deg; joints [-2.08, 63.24, -3.25, -159.522, 61.583, 169.923]
  Call Extruder(1162.11106)
  MoveL 5529 to (505.61, 434.78, 96) mm, rotated rx -180 ry 0 rz 160 deg; joints [-2.048, 63.61, -4.04, -159.406, 61.195, 169.738]
  Set speed (18.0 mm/s)
  Call Extruder(1169.73866)
  MoveL 5530 to (508.03, 435.03, 96) mm, rotated rx -180 ry 0 rz 160 deg; joints [-2.005, 63.98, -4.828, -159.276, 60.811, 169.546]
  Set speed (18.0 mm/s)
  Call Extruder(1177.24869)
  MoveL 5531 to (510.4, 435.37, 96) mm, rotated rx -180 ry 0 rz 160 deg; joints [-1.953, 64.346, -5.608, -159.135, 60.435, 169.349]
  Call Extruder(1184.63365)
  MoveL 5532 to (512.71, 435.78, 96) mm, rotated rx 180 ry 0 rz 160 deg; joints [-1.892, 64.708, -6.377, -158.983, 60.066, 169.147]
  Set speed (18.0 mm/s)
  Call Extruder(1192.36493)
  MoveL 5533 to (515.12, 436.31, 96) mm, rotated rx -180 ry 0 rz 160 deg; joints [-1.818, 65.089, -7.182, -158.809, 59.684, 168.928]
  Set speed (18.0 mm/s)
  Call Extruder(1199.83645)
  MoveL 5534 to (517.43, 436.9, 96) mm, rotated rx 180 ry 0 rz 160 deg; joints [-1.736, 65.458, -7.962, -158.629, 59.317, 168.707]
  Call Extruder(1207.46021)
  MoveL 5535 to (519.76, 437.59, 96) mm, rotated rx 180 ry 0 rz 160 deg; joints [-1.643, 65.836, -8.757, -158.431, 58.947, 168.475]
  Set speed (18.0 mm/s)
  Call Extruder(1215.09271)
  MoveL 5536 to (522.07, 438.37, 96) mm, rotated rx 180 ry 0 rz 160 deg; joints [-1.54, 66.213, -9.551, -158.22, 58.581, 168.234]
  Set speed (18.0 mm/s)
  Call Extruder(1222.46670)
  MoveL 5537 to (524.26, 439.2, 96) mm, rotated rx 180 ry 0 rz 160 deg; joints [-1.433, 66.577, -10.315, -158.005, 58.232, 167.994]
  Set speed (18.0 mm/s)
  Call Extruder(1230.22647)
  MoveL 5538 to (526.54, 440.16, 96) mm, rotated rx 180 ry 0 rz 160 deg; joints [-1.31, 66.96, -11.116, -157.766, 57.87, 167.734]
  Set speed (18.0 mm/s)
  Call Extruder(1237.78738)
  MoveL 5539 to (528.72, 441.17, 96) mm, rotated rx 180 ry 0 rz 160 deg; joints [-1.183, 67.331, -11.892, -157.521, 57.523, 167.473]
  Set speed (18.0 mm/s)
  Call Extruder(1245.26691)
  MoveL 5540 to (530.85, 442.26, 96) mm, rotated rx -180 ry 0 rz 160 deg; joints [-1.048, 67.696, -12.654, -157.267, 57.186, 167.208]
  Set speed (18.0 mm/s)
  Call Extruder(1252.91800)
  MoveL 5541 to (532.98, 443.45, 96) mm, rotated rx -180 ry 0 rz 160 deg; joints [-0.902, 68.067, -13.427, -156.996, 56.848, 166.929]
  Set speed (18.0 mm/s)
  Call Extruder(1260.25642)
  MoveL 5542 to (534.97, 444.66, 96) mm, rotated rx 180 ry 0 rz 160 deg; joints [-0.755, 68.421, -14.162, -156.726, 56.532, 166.656]
  Set speed (18.0 mm/s)
  Call Extruder(1268.03885)
  MoveL 5543 to (537.04, 446.03, 96) mm, rotated rx 180 ry 0 rz 160 deg; joints [-0.591, 68.792, -14.932, -156.429, 56.204, 166.359]
  Set speed (18.0 mm/s)
  Call Extruder(1275.51458)
  MoveL 5544 to (538.99, 447.41, 96) mm, rotated rx 180 ry 0 rz 160 deg; joints [-0.426, 69.145, -15.663, -156.134, 55.897, 166.068]
  Set speed (18.0 mm/s)
  Call Extruder(1283.15752)
  MoveL 5545 to (540.92, 448.9, 96) mm, rotated rx -180 ry 0 rz 160 deg; joints [-0.251, 69.501, -16.399, -155.823, 55.592, 165.765]
  Set speed (18.0 mm/s)
  Call Extruder(1290.52910)
  MoveL 5546 to (542.72, 450.4, 96) mm, rotated rx 180 ry 0 rz 160 deg; joints [-0.075, 69.84, -17.098, -155.514, 55.308, 165.468]
  Call Extruder(1298.28746)
  MoveL 5547 to (544.57, 452.05, 96) mm, rotated rx -180 ry 0 rz 160 deg; joints [0.117, 70.19, -17.82, -155.18, 55.019, 165.15]
  Set speed (18.0 mm/s)
  Call Extruder(1305.79661)
  MoveL 5548 to (546.29, 453.71, 96) mm, rotated rx 180 ry 0 rz 160 deg; joints [0.308, 70.523, -18.505, -154.849, 54.749, 164.838]
  Call Extruder(1309.93007)
  MoveL 5549 to (547.21, 454.65, 96) mm, rotated rx 180 ry 0 rz 160 deg; joints [0.416, 70.703, -18.876, -154.664, 54.605, 164.665]
  Set speed (18.0 mm/s)
  Call Extruder(1314.10222)
  MoveL 5550 to (548.12, 455.62, 96) mm, rotated rx 180 ry 0 rz 160 deg; joints [0.527, 70.883, -19.245, -154.475, 54.464, 164.489]
  Set speed (18.0 mm/s)
  Call Extruder(1318.35507)
  MoveL 5551 to (549.03, 456.63, 96) mm, rotated rx 180 ry 0 rz 160 deg; joints [0.642, 71.064, -19.616, -154.28, 54.323, 164.308]
  Set speed (18.0 mm/s)
  Call Extruder(1322.49002)
  MoveL 5552 to (549.89, 457.62, 96) mm, rotated rx 180 ry 0 rz 160 deg; joints [0.755, 71.237, -19.971, -154.089, 54.19, 164.132]
  Call Extruder(1326.70054)
  MoveL 5553 to (550.75, 458.65, 96) mm, rotated rx -180 ry 0 rz 160 deg; joints [0.872, 71.412, -20.328, -153.892, 54.058, 163.952]
  Call Extruder(1330.92934)
  MoveL 5554 to (551.59, 459.71, 96) mm, rotated rx -180 ry 0 rz 160 deg; joints [0.991, 71.584, -20.681, -153.693, 53.929, 163.77]
  Set speed (18.0 mm/s)
  Call Extruder(1335.10021)
  MoveL 5555 to (552.4, 460.76, 96) mm, rotated rx 180 ry 0 rz 160 deg; joints [1.11, 71.751, -21.022, -153.495, 53.806, 163.591]
  Call Extruder(1339.28682)
  MoveL 5556 to (553.19, 461.84, 96) mm, rotated rx -180 ry 0 rz 160 deg; joints [1.231, 71.916, -21.36, -153.294, 53.686, 163.41]
  Set speed (18.0 mm/s)
  Call Extruder(1343.55647)
  MoveL 5557 to (553.97, 462.95, 96) mm, rotated rx 180 ry 0 rz 160 deg; joints [1.356, 72.081, -21.697, -153.089, 53.568, 163.225]
  Call Extruder(1347.79272)
  MoveL 5558 to (554.73, 464.07, 96) mm, rotated rx 180 ry 0 rz 160 deg; joints [1.481, 72.242, -22.026, -152.883, 53.456, 163.042]
  Set speed (18.0 mm/s)
  Call Extruder(1351.90246)
  MoveL 5559 to (555.43, 465.18, 96) mm, rotated rx 180 ry 0 rz 160 deg; joints [1.604, 72.395, -22.337, -152.683, 53.35, 162.864]
  Set speed (18.0 mm/s)
  Call Extruder(1356.16777)
  MoveL 5560 to (556.14, 466.33, 96) mm, rotated rx 180 ry 0 rz 160 deg; joints [1.733, 72.55, -22.653, -152.474, 53.246, 162.68]
  Set speed (18.0 mm/s)
  Call Extruder(1360.29494)
  MoveL 5561 to (556.81, 467.47, 96) mm, rotated rx 180 ry 0 rz 160 deg; joints [1.859, 72.696, -22.953, -152.271, 53.148, 162.502]
  Call Extruder(1365.79411)
  MoveL 5562 to (557.66, 469, 96) mm, rotated rx -180 ry 0 rz 160 deg; joints [2.029, 72.887, -23.341, -151.999, 53.025, 162.265]
  Call Extruder(1368.71238)
  MoveL 5563 to (558.09, 469.82, 96) mm, rotated rx -180 ry 0 rz 160 deg; joints [2.12, 72.985, -23.541, -151.855, 52.963, 162.14]
  Set speed (18.0 mm/s)
  Call Extruder(1372.89590)
  MoveL 5564 to (558.7, 471.01, 96) mm, rotated rx -180 ry 0 rz 160 deg; joints [2.251, 73.124, -23.822, -151.647, 52.877, 161.96]
  Set speed (18.0 mm/s)
  Call Extruder(1378.25988)
  MoveL 5565 to (559.43, 472.55, 96) mm, rotated rx 180 ry 0 rz 160 deg; joints [2.421, 73.295, -24.17, -151.38, 52.775, 161.732]
  Set speed (18.0 mm/s)
  Call Extruder(1381.39111)
  MoveL 5566 to (559.84, 473.46, 96) mm, rotated rx 180 ry 0 rz 160 deg; joints [2.521, 73.392, -24.367, -151.224, 52.719, 161.599]
  Set speed (18.0 mm/s)
  Call Extruder(1385.62571)
  MoveL 5567 to (560.37, 474.7, 96) mm, rotated rx -180 ry 0 rz 160 deg; joints [2.658, 73.518, -24.624, -151.013, 52.648, 161.421]
  Set speed (18.0 mm/s)
  Call Extruder(1389.71450)
  MoveL 5568 to (560.87, 475.9, 96) mm, rotated rx -180 ry 0 rz 160 deg; joints [2.79, 73.639, -24.869, -150.81, 52.582, 161.25]
  Set speed (18.0 mm/s)
  Call Extruder(1398.15308)
  MoveL 5569 to (561.81, 478.42, 96) mm, rotated rx -180 ry 0 rz 160 deg; joints [3.067, 73.873, -25.343, -150.389, 52.462, 160.9]
  Set speed (18.0 mm/s)
  Call Extruder(1402.43246)
  MoveL 5570 to (562.23, 479.72, 96) mm, rotated rx 180 ry 0 rz 160 deg; joints [3.208, 73.983, -25.566, -150.177, 52.41, 160.727]
  Call Extruder(1406.56607)
  MoveL 5571 to (562.63, 480.97, 96) mm, rotated rx 180 ry 0 rz 160 deg; joints [3.346, 74.087, -25.778, -149.972, 52.363, 160.559]
  Call Extruder(1410.85993)
  MoveL 5572 to (563.01, 482.28, 96) mm, rotated rx -180 ry 0 rz 160 deg; joints [3.49, 74.189, -25.984, -149.761, 52.321, 160.388]
  Set speed (18.0 mm/s)
  Call Extruder(1415.04946)
  MoveL 5573 to (563.37, 483.57, 96) mm, rotated rx 180 ry 0 rz 160 deg; joints [3.63, 74.286, -26.181, -149.554, 52.282, 160.222]
  Set speed (18.0 mm/s)
  Call Extruder(1423.40558)
  MoveL 5574 to (563.99, 486.16, 96) mm, rotated rx -180 ry 0 rz 160 deg; joints [3.914, 74.463, -26.539, -149.146, 52.223, 159.899]
  Call Extruder(1431.84070)
  MoveL 5575 to (564.5, 488.8, 96) mm, rotated rx 180 ry 0 rz 160 deg; joints [4.203, 74.621, -26.859, -148.738, 52.185, 159.584]
  Call Extruder(1440.23685)
  MoveL 5576 to (564.9, 491.44, 96) mm, rotated rx -180 ry 0 rz 160 deg; joints [4.492, 74.759, -27.138, -148.338, 52.166, 159.28]
  Set speed (18.0 mm/s)
  Call Extruder(1448.72489)
  MoveL 5577 to (565.2, 494.13, 96) mm, rotated rx 180 ry 0 rz 160 deg; joints [4.787, 74.877, -27.376, -147.939, 52.169, 158.985]
  Call Extruder(1457.03454)
  MoveL 5578 to (565.39, 496.77, 96) mm, rotated rx -180 ry 0 rz 160 deg; joints [5.078, 74.972, -27.567, -147.556, 52.192, 158.71]
  Call Extruder(1465.42765)
  MoveL 5579 to (565.46, 499.45, 96) mm, rotated rx -180 ry 0 rz 160 deg; joints [5.372, 75.046, -27.716, -147.178, 52.237, 158.446]
  Set speed (18.0 mm/s)
  Call Extruder(1473.71297)
  MoveL 5580 to (565.43, 502.09, 96) mm, rotated rx -180 ry 0 rz 160 deg; joints [5.664, 75.098, -27.821, -146.813, 52.3, 158.2]
  Set speed (18.0 mm/s)
  Call Extruder(1482.22457)
  MoveL 5581 to (565.29, 504.8, 96) mm, rotated rx 180 ry 0 rz 160 deg; joints [5.964, 75.128, -27.883, -146.448, 52.386, 157.964]
  Call Extruder(1490.54118)
  MoveL 5582 to (565.04, 507.44, 96) mm, rotated rx -180 ry 0 rz 160 deg; joints [6.258, 75.136, -27.899, -146.102, 52.49, 157.749]
  Set speed (18.0 mm/s)
  Call Extruder(1499.11826)
  MoveL 5583 to (564.67, 510.15, 96) mm, rotated rx -180 ry 0 rz 160 deg; joints [6.56, 75.122, -27.869, -145.756, 52.617, 157.545]
  Set speed (18.0 mm/s)
  Call Extruder(1507.34108)
  MoveL 5584 to (564.22, 512.73, 96) mm, rotated rx -180 ry 0 rz 160 deg; joints [6.85, 75.086, -27.798, -145.434, 52.758, 157.366]
  Call Extruder(1515.87836)
  MoveL 5585 to (563.63, 515.39, 96) mm, rotated rx -180 ry 0 rz 160 deg; joints [7.151, 75.027, -27.678, -145.113, 52.924, 157.2]
  Set speed (18.0 mm/s)
  Call Extruder(1520.05503)
  MoveL 5586 to (563.3, 516.68, 96) mm, rotated rx -180 ry 0 rz 160 deg; joints [7.297, 74.988, -27.6, -144.961, 53.013, 157.126]
  Call Extruder(1524.16136)
  MoveL 5587 to (562.96, 517.94, 96) mm, rotated rx 180 ry 0 rz 160 deg; joints [7.441, 74.948, -27.518, -144.813, 53.103, 157.056]
  Set speed (18.0 mm/s)
  Call Extruder(1528.45788)
  MoveL 5588 to (562.56, 519.25, 96) mm, rotated rx 180 ry 0 rz 160 deg; joints [7.59, 74.897, -27.416, -144.663, 53.204, 156.99]
  Set speed (18.0 mm/s)
  Call Extruder(1532.54634)
  MoveL 5589 to (562.17, 520.49, 96) mm, rotated rx -180 ry 0 rz 160 deg; joints [7.733, 74.846, -27.313, -144.522, 53.301, 156.93]
  Set speed (18.0 mm/s)
  Call Extruder(1536.86085)
  MoveL 5590 to (561.72, 521.79, 96) mm, rotated rx -180 ry 0 rz 160 deg; joints [7.882, 74.784, -27.188, -144.378, 53.411, 156.873]
  Set speed (18.0 mm/s)
  Call Extruder(1540.98649)
  MoveL 5591 to (561.28, 523.03, 96) mm, rotated rx -180 ry 0 rz 160 deg; joints [8.025, 74.723, -27.064, -144.242, 53.518, 156.822]
  Set speed (18.0 mm/s)
  Call Extruder(1545.28612)
  MoveL 5592 to (560.78, 524.3, 96) mm, rotated rx -180 ry 0 rz 160 deg; joints [8.173, 74.652, -26.92, -144.104, 53.636, 156.774]
  Set speed (18.0 mm/s)
  Call Extruder(1549.39147)
  MoveL 5593 to (560.29, 525.51, 96) mm, rotated rx -180 ry 0 rz 160 deg; joints [8.314, 74.58, -26.776, -143.974, 53.75, 156.732]
  Set speed (18.0 mm/s)
  Call Extruder(1557.76532)
  MoveL 5594 to (559.2, 527.95, 96) mm, rotated rx -180 ry 0 rz 160 deg; joints [8.601, 74.417, -26.446, -143.721, 53.998, 156.662]
  Set speed (18.0 mm/s)
  Call Extruder(1562.02091)
  MoveL 5595 to (558.61, 529.17, 96) mm, rotated rx 180 ry 0 rz 160 deg; joints [8.745, 74.327, -26.263, -143.597, 54.13, 156.633]
  Set speed (18.0 mm/s)
  Call Extruder(1566.28107)
  MoveL 5596 to (557.99, 530.38, 96) mm, rotated rx 180 ry 0 rz 160 deg; joints [8.889, 74.232, -26.071, -143.476, 54.265, 156.609]
  Set speed (18.0 mm/s)
  Call Extruder(1570.49081)
  MoveL 5597 to (557.35, 531.56, 96) mm, rotated rx 180 ry 0 rz 160 deg; joints [9.03, 74.133, -25.87, -143.359, 54.403, 156.591]
  Call Extruder(0.00000)
  Set speed (18.0 mm/s)
  Call Extruder(4.15341)
  MoveL 5598 to (556.71, 532.72, 96) mm, rotated rx 180 ry 0 rz 160 deg; joints [9.169, 74.031, -25.664, -143.247, 54.542, 156.576]
  Set speed (18.0 mm/s)
  Call Extruder(9.22205)
  MoveL 5599 to (555.88, 534.1, 96) mm, rotated rx -180 ry 0 rz 160 deg; joints [9.337, 73.9, -25.399, -143.115, 54.716, 156.566]
  Set speed (18.0 mm/s)
  Call Extruder(12.51098)
  MoveL 5600 to (555.33, 534.99, 96) mm, rotated rx 180 ry 0 rz 160 deg; joints [9.446, 73.812, -25.22, -143.032, 54.832, 156.562]
  Set speed (18.0 mm/s)
  Call Extruder(16.73631)
  MoveL 5601 to (554.6, 536.12, 96) mm, rotated rx -180 ry 0 rz 160 deg; joints [9.584, 73.694, -24.981, -142.928, 54.984, 156.562]
  Set speed (18.0 mm/s)
  Call Extruder(20.95695)
  MoveL 5602 to (553.84, 537.24, 96) mm, rotated rx -180 ry 0 rz 160 deg; joints [9.722, 73.573, -24.735, -142.827, 55.138, 156.566]
  Call Extruder(25.13568)
  MoveL 5603 to (553.07, 538.33, 96) mm, rotated rx 180 ry 0 rz 160 deg; joints [9.857, 73.448, -24.482, -142.73, 55.294, 156.574]
  Call Extruder(29.35569)
  MoveL 5604 to (552.27, 539.41, 96) mm, rotated rx -180 ry 0 rz 160 deg; joints [9.992, 73.319, -24.219, -142.635, 55.454, 156.587]
  Set speed (18.0 mm/s)
  Call Extruder(34.51361)
  MoveL 5605 to (551.27, 540.71, 96) mm, rotated rx -180 ry 0 rz 160 deg; joints [10.156, 73.155, -23.886, -142.523, 55.653, 156.608]
  Set speed (18.0 mm/s)
  Call Extruder(37.79040)
  MoveL 5606 to (550.61, 541.52, 96) mm, rotated rx -180 ry 0 rz 160 deg; joints [10.259, 73.047, -23.667, -142.454, 55.783, 156.626]
  Set speed (18.0 mm/s)
  Call Extruder(42.04231)
  MoveL 5607 to (549.74, 542.56, 96) mm, rotated rx 180 ry 0 rz 160 deg; joints [10.392, 72.905, -23.377, -142.368, 55.952, 156.652]
  Call Extruder(46.12704)
  MoveL 5608 to (548.88, 543.54, 96) mm, rotated rx -180 ry 0 rz 160 deg; joints [10.519, 72.764, -23.091, -142.288, 56.118, 156.681]
  Set speed (18.0 mm/s)
  Call Extruder(50.35369)
  MoveL 5609 to (547.98, 544.54, 96) mm, rotated rx -180 ry 0 rz 160 deg; joints [10.649, 72.616, -22.789, -142.207, 56.291, 156.714]
  Set speed (18.0 mm/s)
  Call Extruder(54.53971)
  MoveL 5610 to (547.06, 545.51, 96) mm, rotated rx -180 ry 0 rz 160 deg; joints [10.776, 72.465, -22.481, -142.131, 56.465, 156.752]
  Call Extruder(58.77546)
  MoveL 5611 to (546.11, 546.47, 96) mm, rotated rx 180 ry 0 rz 160 deg; joints [10.903, 72.309, -22.163, -142.057, 56.643, 156.794]
  Set speed (18.0 mm/s)
  Call Extruder(62.92467)
  MoveL 5612 to (545.17, 547.39, 96) mm, rotated rx 180 ry 0 rz 160 deg; joints [11.026, 72.153, -21.844, -141.987, 56.819, 156.839]
  Call Extruder(67.12914)
  MoveL 5613 to (544.19, 548.3, 96) mm, rotated rx -180 ry 0 rz 160 deg; joints [11.15, 71.992, -21.515, -141.918, 57, 156.889]
  Set speed (18.0 mm/s)
  Call Extruder(71.37592)
  MoveL 5614 to (543.18, 549.21, 96) mm, rotated rx -180 ry 0 rz 160 deg; joints [11.273, 71.826, -21.177, -141.852, 57.184, 156.942]
  Set speed (18.0 mm/s)
  Call Extruder(75.55710)
  MoveL 5615 to (542.17, 550.07, 96) mm, rotated rx -180 ry 0 rz 160 deg; joints [11.393, 71.66, -20.836, -141.79, 57.368, 157]
  Call Extruder(79.83394)
  MoveL 5616 to (541.12, 550.94, 96) mm, rotated rx 180 ry 0 rz 160 deg; joints [11.514, 71.487, -20.483, -141.729, 57.558, 157.061]
  Call Extruder(83.40569)
  MoveL 5617 to (540.22, 551.65, 96) mm, rotated rx 180 ry 0 rz 160 deg; joints [11.614, 71.34, -20.182, -141.681, 57.717, 157.116]
  Set speed (18.0 mm/s)
  Call Extruder(88.11694)
  MoveL 5618 to (539.03, 552.56, 96) mm, rotated rx 180 ry 0 rz 160 deg; joints [11.744, 71.144, -19.78, -141.62, 57.929, 157.191]
  Set speed (18.0 mm/s)
  Call Extruder(92.42086)
  MoveL 5619 to (537.92, 553.36, 96) mm, rotated rx -180 ry 0 rz 160 deg; joints [11.861, 70.962, -19.407, -141.567, 58.124, 157.264]
  Set speed (18.0 mm/s)
  Call Extruder(96.53433)
  MoveL 5620 to (536.84, 554.11, 96) mm, rotated rx 180 ry 0 rz 160 deg; joints [11.971, 70.786, -19.045, -141.519, 58.312, 157.337]
  Set speed (18.0 mm/s)
  Call Extruder(100.82624)
  MoveL 5621 to (535.7, 554.87, 96) mm, rotated rx 180 ry 0 rz 160 deg; joints [12.084, 70.6, -18.663, -141.472, 58.509, 157.416]
  Call Extruder(104.99382)
  MoveL 5622 to (534.58, 555.58, 96) mm, rotated rx 180 ry 0 rz 160 deg; joints [12.192, 70.417, -18.286, -141.429, 58.701, 157.497]
  Call Extruder(109.19450)
  MoveL 5623 to (533.44, 556.28, 96) mm, rotated rx 180 ry 0 rz 160 deg; joints [12.298, 70.23, -17.902, -141.388, 58.897, 157.581]
  Call Extruder(113.44391)
  MoveL 5624 to (532.27, 556.96, 96) mm, rotated rx 180 ry 0 rz 160 deg; joints [12.405, 70.04, -17.51, -141.349, 59.095, 157.669]
  Set speed (18.0 mm/s)
  Call Extruder(117.00025)
  MoveL 5625 to (531.28, 557.51, 96) mm, rotated rx -180 ry 0 rz 160 deg; joints [12.492, 69.879, -17.178, -141.318, 59.261, 157.745]
  Set speed (18.0 mm/s)
  Call Extruder(122.98830)
  MoveL 5626 to (529.59, 558.4, 96) mm, rotated rx -180 ry 0 rz 160 deg; joints [12.636, 69.606, -16.615, -141.271, 59.542, 157.877]
  Set speed (18.0 mm/s)
  Call Extruder(126.04935)
  MoveL 5627 to (528.72, 558.83, 96) mm, rotated rx 180 ry 0 rz 160 deg; joints [12.708, 69.464, -16.321, -141.25, 59.687, 157.948]
  Set speed (18.0 mm/s)
  Call Extruder(130.13399)
  MoveL 5628 to (527.54, 559.39, 96) mm, rotated rx 180 ry 0 rz 160 deg; joints [12.802, 69.274, -15.929, -141.223, 59.881, 158.044]
  Set speed (18.0 mm/s)
  Call Extruder(134.44620)
  MoveL 5629 to (526.29, 559.95, 96) mm, rotated rx 180 ry 0 rz 160 deg; joints [12.899, 69.071, -15.51, -141.197, 60.085, 158.148]
  Call Extruder(138.79917)
  MoveL 5630 to (525.01, 560.5, 96) mm, rotated rx 180 ry 0 rz 160 deg; joints [12.995, 68.867, -15.087, -141.173, 60.292, 158.255]
  Set speed (18.0 mm/s)
  Call Extruder(146.86266)
  MoveL 5631 to (522.62, 561.43, 96) mm, rotated rx 180 ry 0 rz 160 deg; joints [13.166, 68.483, -14.29, -141.136, 60.676, 158.463]
  Set speed (18.0 mm/s)
  Call Extruder(151.30260)
  MoveL 5632 to (521.29, 561.9, 96) mm, rotated rx -180 ry 0 rz 160 deg; joints [13.256, 68.269, -13.847, -141.121, 60.888, 158.581]
  Call Extruder(155.34951)
  MoveL 5633 to (520.07, 562.31, 96) mm, rotated rx 180 ry 0 rz 160 deg; joints [13.337, 68.075, -13.442, -141.108, 61.081, 158.69]
  Call Extruder(159.64920)
  MoveL 5634 to (518.76, 562.71, 96) mm, rotated rx 180 ry 0 rz 160 deg; joints [13.419, 67.866, -13.008, -141.098, 61.286, 158.809]
  Set speed (18.0 mm/s)
  Call Extruder(163.75289)
  MoveL 5635 to (517.5, 563.08, 96) mm, rotated rx -180 ry 0 rz 160 deg; joints [13.497, 67.667, -12.593, -141.09, 61.482, 158.924]
  Set speed (18.0 mm/s)
  Call Extruder(167.55890)
  MoveL 5636 to (516.33, 563.39, 96) mm, rotated rx 180 ry 0 rz 160 deg; joints [13.565, 67.481, -12.206, -141.086, 61.663, 159.034]
  Call Extruder(172.13117)
  MoveL 5637 to (514.92, 563.74, 96) mm, rotated rx -180 ry 0 rz 160 deg; joints [13.646, 67.258, -11.74, -141.082, 61.881, 159.166]
  Set speed (18.0 mm/s)
  Call Extruder(180.69190)
  MoveL 5638 to (512.25, 564.31, 96) mm, rotated rx -180 ry 0 rz 160 deg; joints [13.789, 66.837, -10.86, -141.084, 62.289, 159.422]
  Call Extruder(189.14449)
  MoveL 5639 to (509.59, 564.76, 96) mm, rotated rx -180 ry 0 rz 160 deg; joints [13.918, 66.42, -9.985, -141.097, 62.69, 159.683]
  Set speed (18.0 mm/s)
  Call Extruder(197.46906)
  MoveL 5640 to (506.96, 565.09, 96) mm, rotated rx 180 ry 0 rz 160 deg; joints [14.035, 66.008, -9.12, -141.119, 63.083, 159.946]
  Call Extruder(205.91501)
  MoveL 5641 to (504.28, 565.32, 96) mm, rotated rx 180 ry 0 rz 160 deg; joints [14.142, 65.59, -8.24, -141.152, 63.479, 160.22]
  Set speed (18.0 mm/s)
  Call Extruder(214.35757)
  MoveL 5642 to (501.59, 565.45, 96) mm, rotated rx -180 ry 0 rz 160 deg; joints [14.238, 65.173, -7.36, -141.196, 63.872, 160.5]
  Call Extruder(222.57500)
  MoveL 5643 to (498.97, 565.46, 96) mm, rotated rx 180 ry 0 rz 160 deg; joints [14.319, 64.768, -6.504, -141.248, 64.251, 160.777]
  Set speed (10.0 mm/s)
  MoveL 5644 to (498.97, 565.46, 100) mm, rotated rx 180 ry 0 rz 160 deg; joints [14.319, 64.132, -6.205, -141.146, 63.988, 160.542]
  Set speed (120.0 mm/s)
  MoveL 5645 to (498.98, 565.21, 100) mm, rotated rx 180 ry 0 rz 160 deg; joints [14.289, 64.123, -6.186, -141.179, 63.986, 160.562]
  Set speed (17.9 mm/s)
  Call Extruder(231.15008)
  MoveL 5646 to (496.26, 565.11, 100) mm, rotated rx 180 ry 0 rz 160 deg; joints [14.361, 63.702, -5.3, -141.246, 64.373, 160.854]
  Set speed (17.9 mm/s)
  Call Extruder(239.58198)
  MoveL 5647 to (493.59, 564.91, 100) mm, rotated rx -180 ry 0 rz 160 deg; joints [14.419, 63.291, -4.431, -141.321, 64.748, 161.145]
  Set speed (17.9 mm/s)
  Call Extruder(247.92902)
  MoveL 5648 to (490.97, 564.59, 100) mm, rotated rx 180 ry 0 rz 160 deg; joints [14.463, 62.887, -3.575, -141.407, 65.116, 161.437]
  Set speed (17.9 mm/s)
  Call Extruder(256.24918)
  MoveL 5649 to (488.36, 564.17, 100) mm, rotated rx -180 ry 0 rz 160 deg; joints [14.494, 62.487, -2.725, -141.504, 65.477, 161.732]
  Call Extruder(264.84537)
  MoveL 5650 to (485.69, 563.63, 100) mm, rotated rx -180 ry 0 rz 160 deg; joints [14.512, 62.078, -1.854, -141.614, 65.845, 162.039]
  Set speed (17.9 mm/s)
  Call Extruder(272.97422)
  MoveL 5651 to (483.18, 563.02, 100) mm, rotated rx 180 ry 0 rz 160 deg; joints [14.516, 61.696, -1.038, -141.73, 66.187, 162.332]
  Set speed (17.9 mm/s)
  Call Extruder(277.79601)
  MoveL 5652 to (481.71, 562.6, 100) mm, rotated rx -180 ry 0 rz 160 deg; joints [14.512, 61.471, -0.557, -141.804, 66.386, 162.506]
  Set speed (17.9 mm/s)
  Call Extruder(281.54458)
  MoveL 5653 to (480.58, 562.26, 100) mm, rotated rx 180 ry 0 rz 160 deg; joints [14.506, 61.298, -0.186, -141.863, 66.54, 162.642]
  Call Extruder(285.79940)
  MoveL 5654 to (479.3, 561.84, 100) mm, rotated rx 180 ry 0 rz 160 deg; joints [14.495, 61.103, 0.233, -141.934, 66.713, 162.797]
  Set speed (17.9 mm/s)
  Call Extruder(289.98518)
  MoveL 5655 to (478.04, 561.41, 100) mm, rotated rx -180 ry 0 rz 160 deg; joints [14.482, 60.912, 0.642, -142.005, 66.881, 162.949]
  Set speed (17.9 mm/s)
  Call Extruder(298.25652)
  MoveL 5656 to (475.59, 560.48, 100) mm, rotated rx 180 ry 0 rz 160 deg; joints [14.444, 60.539, 1.445, -142.157, 67.209, 163.251]
  Set speed (17.9 mm/s)
  Call Extruder(302.66436)
  MoveL 5657 to (474.3, 559.94, 100) mm, rotated rx -180 ry 0 rz 160 deg; joints [14.418, 60.343, 1.868, -142.242, 67.38, 163.412]
  Set speed (17.9 mm/s)
  Call Extruder(307.22686)
  MoveL 5658 to (472.98, 559.36, 100) mm, rotated rx 180 ry 0 rz 160 deg; joints [14.388, 60.141, 2.302, -142.333, 67.556, 163.579]
  Set speed (17.9 mm/s)
  Call Extruder(311.01241)
  MoveL 5659 to (471.89, 558.86, 100) mm, rotated rx -180 ry 0 rz 160 deg; joints [14.358, 59.976, 2.66, -142.411, 67.7, 163.717]
  Set speed (17.9 mm/s)
  Call Extruder(315.19066)
  MoveL 5660 to (470.7, 558.27, 100) mm, rotated rx -180 ry 0 rz 160 deg; joints [14.323, 59.795, 3.051, -142.501, 67.858, 163.87]
  Set speed (17.9 mm/s)
  Call Extruder(319.89323)
  MoveL 5661 to (469.38, 557.58, 100) mm, rotated rx 180 ry 0 rz 160 deg; joints [14.278, 59.594, 3.488, -142.605, 68.032, 164.042]
  Set speed (17.9 mm/s)
  Call Extruder(323.57935)
  MoveL 5662 to (468.35, 557.03, 100) mm, rotated rx -180 ry 0 rz 160 deg; joints [14.24, 59.437, 3.827, -142.69, 68.167, 164.176]
  Set speed (17.9 mm/s)
  Call Extruder(328.92736)
  MoveL 5663 to (466.88, 556.19, 100) mm, rotated rx 180 ry 0 rz 160 deg; joints [14.179, 59.213, 4.315, -142.816, 68.36, 164.371]
  Set speed (17.9 mm/s)
  Call Extruder(332.06704)
  MoveL 5664 to (466.02, 555.67, 100) mm, rotated rx 180 ry 0 rz 160 deg; joints [14.14, 59.083, 4.597, -142.892, 68.471, 164.485]
  Set speed (17.9 mm/s)
  Call Extruder(336.73766)
  MoveL 5665 to (464.77, 554.89, 100) mm, rotated rx 180 ry 0 rz 160 deg; joints [14.079, 58.892, 5.014, -143.009, 68.635, 164.654]
  Set speed (17.9 mm/s)
  Call Extruder(339.83915)
  MoveL 5666 to (463.94, 554.35, 100) mm, rotated rx -180 ry 0 rz 160 deg; joints [14.036, 58.767, 5.288, -143.088, 68.742, 164.766]
  Set speed (17.9 mm/s)
  Call Extruder(344.69337)
  MoveL 5667 to (462.67, 553.49, 100) mm, rotated rx -180 ry 0 rz 160 deg; joints [13.965, 58.573, 5.711, -143.216, 68.907, 164.94]
  Set speed (17.9 mm/s)
  Call Extruder(348.92569)
  MoveL 5668 to (461.58, 552.71, 100) mm, rotated rx 180 ry 0 rz 160 deg; joints [13.898, 58.406, 6.076, -143.33, 69.049, 165.092]
  Set speed (17.9 mm/s)
  Call Extruder(354.01294)
  MoveL 5669 to (460.29, 551.74, 100) mm, rotated rx -180 ry 0 rz 160 deg; joints [13.813, 58.209, 6.509, -143.472, 69.216, 165.274]
  Set speed (17.9 mm/s)
  Call Extruder(357.10867)
  MoveL 5670 to (459.51, 551.14, 100) mm, rotated rx 180 ry 0 rz 160 deg; joints [13.758, 58.09, 6.769, -143.56, 69.316, 165.383]
  Set speed (17.9 mm/s)
  Call Extruder(361.47808)
  MoveL 5671 to (458.44, 550.27, 100) mm, rotated rx 180 ry 0 rz 160 deg; joints [13.678, 57.925, 7.131, -143.688, 69.455, 165.538]
  Set speed (17.9 mm/s)
  Call Extruder(366.14299)
  MoveL 5672 to (457.31, 549.31, 100) mm, rotated rx 180 ry 0 rz 160 deg; joints [13.587, 57.752, 7.512, -143.827, 69.6, 165.702]
  Call Extruder(369.87590)
  MoveL 5673 to (456.42, 548.52, 100) mm, rotated rx 180 ry 0 rz 160 deg; joints [13.511, 57.616, 7.813, -143.942, 69.714, 165.832]
  Set speed (17.9 mm/s)
  Call Extruder(374.05457)
  MoveL 5674 to (455.44, 547.63, 100) mm, rotated rx -180 ry 0 rz 160 deg; joints [13.423, 57.465, 8.145, -144.073, 69.839, 165.978]
  Set speed (17.9 mm/s)
  Call Extruder(377.46025)
  MoveL 5675 to (454.66, 546.89, 100) mm, rotated rx -180 ry 0 rz 160 deg; joints [13.348, 57.344, 8.412, -144.181, 69.94, 166.095]
  Set speed (17.9 mm/s)
  Call Extruder(382.54318)
  MoveL 5676 to (453.51, 545.75, 100) mm, rotated rx 180 ry 0 rz 160 deg; joints [13.231, 57.167, 8.803, -144.347, 70.086, 166.27]
  Set speed (17.9 mm/s)
  Call Extruder(386.74169)
  MoveL 5677 to (452.59, 544.79, 100) mm, rotated rx 180 ry 0 rz 160 deg; joints [13.131, 57.024, 9.12, -144.487, 70.204, 166.413]
  Set speed (17.9 mm/s)
  Call Extruder(391.10223)
  MoveL 5678 to (451.65, 543.77, 100) mm, rotated rx 180 ry 0 rz 160 deg; joints [13.023, 56.878, 9.444, -144.636, 70.323, 166.56]
  Set speed (17.9 mm/s)
  Call Extruder(395.09515)
